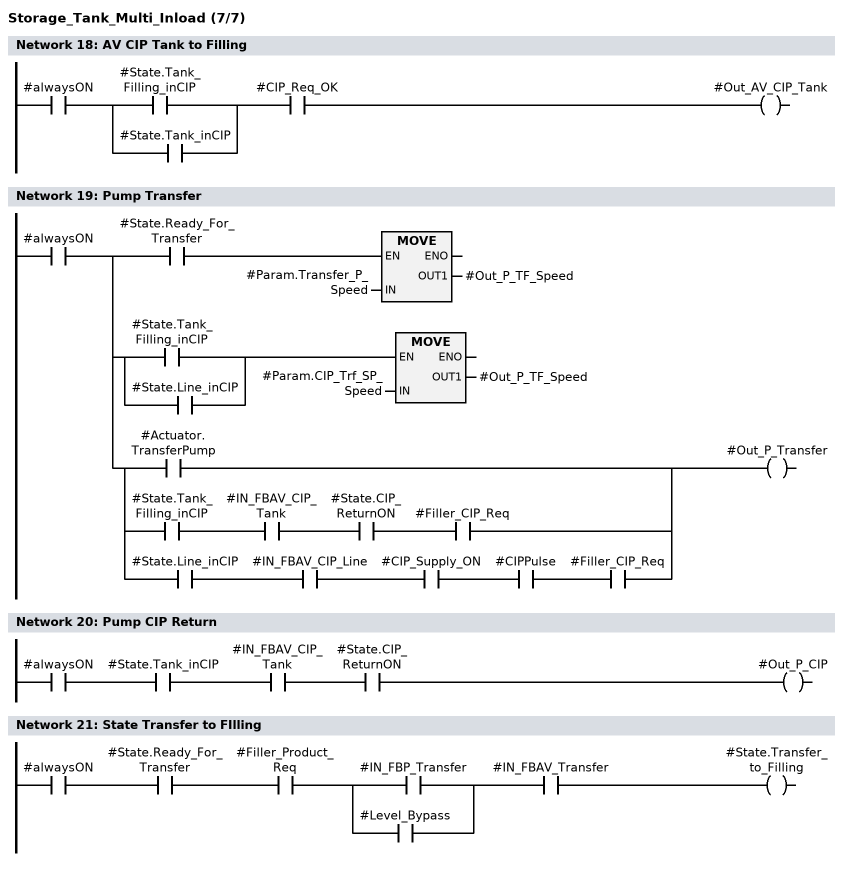
   RUNG wire#powerrail
      Contact( #alwaysON )
      wire#w1
      Contact( #State.Tank_Filling_inCIP )
      wire#w2
      Contact( #CIP_Req_OK )
      Coil( #Out_AV_CIP_Tank )
   END_RUNG
   RUNG wire#w1
      Contact( #State.Tank_inCIP )
   END_RUNG wire#w2
   // the same network as SCL:
   #Out_AV_CIP_Tank := #alwaysON AND (#State.Tank_Filling_inCIP OR #State.Tank_inCIP) AND #CIP_Req_OK;
END_REGION

REGION Network 19: Pump Transfer
   RUNG wire#powerrail
      Contact( #alwaysON )
      wire#w1
      Contact( #State.Ready_For_Transfer )
      Move(in := #Param.Transfer_P_Speed, out1 => #Out_P_TF_Speed)
   END_RUNG
   RUNG wire#w1
      Contact( #State.Tank_Filling_inCIP )
      wire#w2
      Move(in := #Param.CIP_Trf_SP_Speed, out1 => #Out_P_TF_Speed)
   END_RUNG
   RUNG wire#w1
      Contact( #State.Line_inCIP )
   END_RUNG wire#w2
   RUNG wire#w1
      Contact( #Actuator.TransferPump )
      wire#w3
      Coil( #Out_P_Transfer )
   END_RUNG
   RUNG wire#w1
      Contact( #State.Tank_Filling_inCIP )
      Contact( #IN_FBAV_CIP_Tank )
      Contact( #State.CIP_ReturnON )
      Contact( #Filler_CIP_Req )
   END_RUNG wire#w3
   RUNG wire#w1
      Contact( #State.Line_inCIP )
      Contact( #IN_FBAV_CIP_Line )
      Contact( #CIP_Supply_ON )
      Contact( #CIPPulse )
      Contact( #Filler_CIP_Req )
   END_RUNG wire#w3
   // the same network as SCL:
   IF #alwaysON AND #State.Ready_For_Transfer THEN #Out_P_TF_Speed := #Param.Transfer_P_Speed; END_IF;
   IF #alwaysON AND (#State.Tank_Filling_inCIP OR #State.Line_inCIP) THEN
       #Out_P_TF_Speed := #Param.CIP_Trf_SP_Speed;
   END_IF;
   #Out_P_Transfer := #alwaysON AND (#Actuator.TransferPump OR (#State.Tank_Filling_inCIP AND #IN_FBAV_CIP_Tank AND #State.CIP_ReturnON AND #Filler_CIP_Req) OR (#State.Line_inCIP AND #IN_FBAV_CIP_Line AND #CIP_Supply_ON AND #CIPPulse AND #Filler_CIP_Req));
END_REGION

REGION Network 20: Pump CIP Return
   RUNG wire#powerrail
      Contact( #alwaysON )
      Contact( #State.Tank_inCIP )
      Contact( #IN_FBAV_CIP_Tank )
      Contact( #State.CIP_ReturnON )
      Coil( #Out_P_CIP )
   END_RUNG
   // the same network as SCL:
   #Out_P_CIP := #alwaysON AND #State.Tank_inCIP AND #IN_FBAV_CIP_Tank AND #State.CIP_ReturnON;
END_REGION

REGION Network 21: State Transfer to FIlling
   RUNG wire#powerrail
      Contact( #alwaysON )
      Contact( #State.Ready_For_Transfer )
      Contact( #Filler_Product_Req )
      wire#w1
      Contact( #IN_FBP_Transfer )
      wire#w2
      Contact( #IN_FBAV_Transfer )
      Coil( #State.Transfer_to_Filling )
   END_RUNG
   RUNG wire#w1
      Contact( #Level_Bypass )
   END_RUNG wire#w2
   // the same network as SCL:
   #State.Transfer_to_Filling := #alwaysON AND #State.Ready_For_Transfer AND #Filler_Product_Req AND (#IN_FBP_Transfer OR #Level_Bypass) AND #IN_FBAV_Transfer;
END_REGION
END_FUNCTION_BLOCK

FUNCTION "Buffer" : Void   // FC11, LAD
{ S7_Optimized_Access := 'TRUE' }
VERSION : 0.1
// stored: AutoNumber true, IsIECCheckEnabled false, SetENOAutomatically false, UDAEnableTagReadback false
BEGIN

REGION Network 1: BFT 61 Rework 32
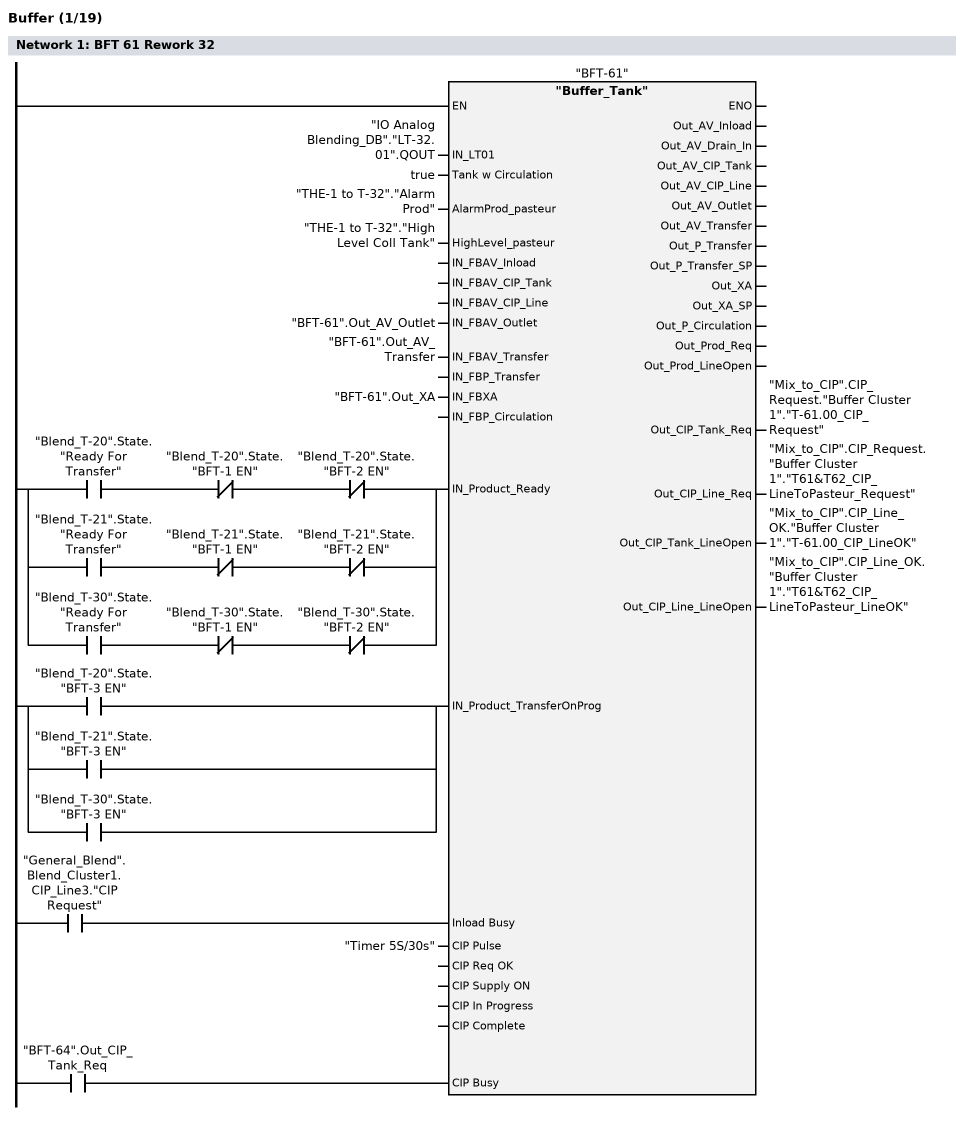
   RUNG wire#powerrail
      "BFT-61"(IN_Product_Ready := wire#w1, IN_Product_TransferOnProg := wire#w2, "Inload Busy" := wire#w3, "CIP Busy" := wire#w4, IN_LT01 := "IO Analog Blending_DB"."LT-32.01".QOUT, "Tank w Circulation" := true, AlarmProd_pasteur := "THE-1 to T-32"."Alarm Prod", HighLevel_pasteur := "THE-1 to T-32"."High Level Coll Tank", IN_FBAV_Inload :=, IN_FBAV_CIP_Tank :=, IN_FBAV_CIP_Line :=, IN_FBAV_Outlet := "BFT-61".Out_AV_Outlet, IN_FBAV_Transfer := "BFT-61".Out_AV_Transfer, IN_FBP_Transfer :=, IN_FBXA := "BFT-61".Out_XA, IN_FBP_Circulation :=, "CIP Pulse" := "Timer 5S/30s", "CIP Req OK" :=, "CIP Supply ON" :=, "CIP In Progress" :=, "CIP Complete" :=, Out_AV_Inload =>, Out_AV_Drain_In =>, Out_AV_CIP_Tank =>, Out_AV_CIP_Line =>, Out_AV_Outlet =>, Out_AV_Transfer =>, Out_P_Transfer =>, Out_P_Transfer_SP =>, Out_XA =>, Out_XA_SP =>, Out_P_Circulation =>, Out_Prod_Req =>, Out_Prod_LineOpen =>, Out_CIP_Tank_Req => "Mix_to_CIP".CIP_Request."Buffer Cluster 1"."T-61.00_CIP_Request", Out_CIP_Line_Req => "Mix_to_CIP".CIP_Request."Buffer Cluster 1"."T61&T62_CIP_LineToPasteur_Request", Out_CIP_Tank_LineOpen => "Mix_to_CIP".CIP_Line_OK."Buffer Cluster 1"."T-61.00_CIP_LineOK", Out_CIP_Line_LineOpen => "Mix_to_CIP".CIP_Line_OK."Buffer Cluster 1"."T61&T62_CIP_LineToPasteur_LineOK")
   END_RUNG
   RUNG wire#powerrail
      Contact( "Blend_T-20".State."Ready For Transfer" )
      I_Contact( "Blend_T-20".State."BFT-1 EN" )
      I_Contact( "Blend_T-20".State."BFT-2 EN" )
   END_RUNG wire#w1
   RUNG wire#powerrail
      Contact( "Blend_T-21".State."Ready For Transfer" )
      I_Contact( "Blend_T-21".State."BFT-1 EN" )
      I_Contact( "Blend_T-21".State."BFT-2 EN" )
   END_RUNG wire#w1
   RUNG wire#powerrail
      Contact( "Blend_T-30".State."Ready For Transfer" )
      I_Contact( "Blend_T-30".State."BFT-1 EN" )
      I_Contact( "Blend_T-30".State."BFT-2 EN" )
   END_RUNG wire#w1
   RUNG wire#powerrail
      Contact( "Blend_T-20".State."BFT-3 EN" )
   END_RUNG wire#w2
   RUNG wire#powerrail
      Contact( "Blend_T-21".State."BFT-3 EN" )
   END_RUNG wire#w2
   RUNG wire#powerrail
      Contact( "Blend_T-30".State."BFT-3 EN" )
   END_RUNG wire#w2
   RUNG wire#powerrail
      Contact( "General_Blend".Blend_Cluster1.CIP_Line3."CIP Request" )
   END_RUNG wire#w3
   RUNG wire#powerrail
      Contact( "BFT-64".Out_CIP_Tank_Req )
   END_RUNG wire#w4
   // the same network as SCL:
   "BFT-61"(IN_LT01 := "IO Analog Blending_DB"."LT-32.01".QOUT,   // "Buffer_Tank"
            "Tank w Circulation" := true,
            AlarmProd_pasteur := "THE-1 to T-32"."Alarm Prod",
            HighLevel_pasteur := "THE-1 to T-32"."High Level Coll Tank",
            IN_FBAV_Outlet := "BFT-61".Out_AV_Outlet,
            IN_FBAV_Transfer := "BFT-61".Out_AV_Transfer,
            IN_FBXA := "BFT-61".Out_XA,
            IN_Product_Ready := ("Blend_T-20".State."Ready For Transfer" AND NOT "Blend_T-20".State."BFT-1 EN" AND NOT "Blend_T-20".State."BFT-2 EN") OR ("Blend_T-21".State."Ready For Transfer" AND NOT "Blend_T-21".State."BFT-1 EN" AND NOT "Blend_T-21".State."BFT-2 EN") OR ("Blend_T-30".State."Ready For Transfer" AND NOT "Blend_T-30".State."BFT-1 EN" AND NOT "Blend_T-30".State."BFT-2 EN"),
            IN_Product_TransferOnProg := "Blend_T-20".State."BFT-3 EN" OR "Blend_T-21".State."BFT-3 EN" OR "Blend_T-30".State."BFT-3 EN",
            "Inload Busy" := "General_Blend".Blend_Cluster1.CIP_Line3."CIP Request",
            "CIP Pulse" := "Timer 5S/30s",
            "CIP Busy" := "BFT-64".Out_CIP_Tank_Req,
            Out_CIP_Tank_Req => "Mix_to_CIP".CIP_Request."Buffer Cluster 1"."T-61.00_CIP_Request",
            Out_CIP_Line_Req => "Mix_to_CIP".CIP_Request."Buffer Cluster 1"."T61&T62_CIP_LineToPasteur_Request",
            Out_CIP_Tank_LineOpen => "Mix_to_CIP".CIP_Line_OK."Buffer Cluster 1"."T-61.00_CIP_LineOK",
            Out_CIP_Line_LineOpen => "Mix_to_CIP".CIP_Line_OK."Buffer Cluster 1"."T61&T62_CIP_LineToPasteur_LineOK");
END_REGION

REGION Network 2: BFT 61 Feedback Instrument
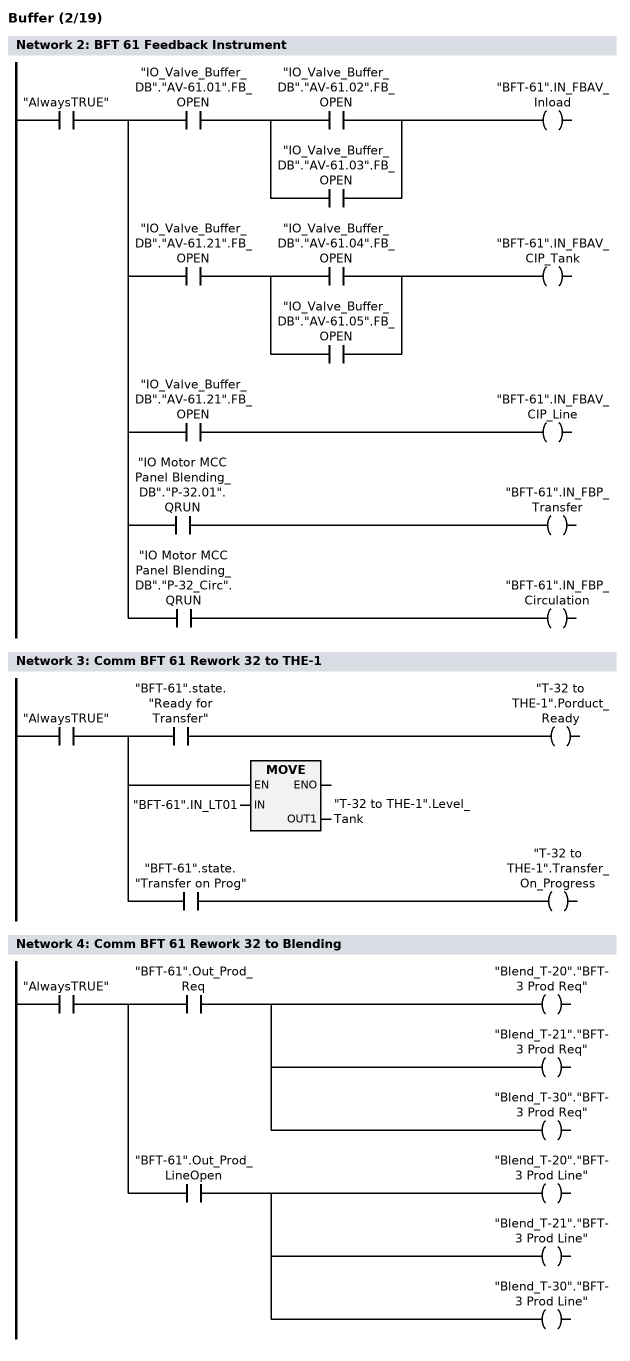
   RUNG wire#powerrail
      Contact( "AlwaysTRUE" )
      wire#w1
      Contact( "IO_Valve_Buffer_DB"."AV-61.01".FB_OPEN )
      wire#w2
      Contact( "IO_Valve_Buffer_DB"."AV-61.02".FB_OPEN )
      wire#w3
      Coil( "BFT-61".IN_FBAV_Inload )
   END_RUNG
   RUNG wire#w2
      Contact( "IO_Valve_Buffer_DB"."AV-61.03".FB_OPEN )
   END_RUNG wire#w3
   RUNG wire#w1
      Contact( "IO_Valve_Buffer_DB"."AV-61.21".FB_OPEN )
      wire#w4
      Contact( "IO_Valve_Buffer_DB"."AV-61.04".FB_OPEN )
      wire#w5
      Coil( "BFT-61".IN_FBAV_CIP_Tank )
   END_RUNG
   RUNG wire#w4
      Contact( "IO_Valve_Buffer_DB"."AV-61.05".FB_OPEN )
   END_RUNG wire#w5
   RUNG wire#w1
      Contact( "IO_Valve_Buffer_DB"."AV-61.21".FB_OPEN )
      Coil( "BFT-61".IN_FBAV_CIP_Line )
   END_RUNG
   RUNG wire#w1
      Contact( "IO Motor MCC Panel Blending_DB"."P-32.01".QRUN )
      Coil( "BFT-61".IN_FBP_Transfer )
   END_RUNG
   RUNG wire#w1
      Contact( "IO Motor MCC Panel Blending_DB"."P-32_Circ".QRUN )
      Coil( "BFT-61".IN_FBP_Circulation )
   END_RUNG
   // the same network as SCL:
   "BFT-61".IN_FBAV_Inload := "AlwaysTRUE" AND "IO_Valve_Buffer_DB"."AV-61.01".FB_OPEN AND ("IO_Valve_Buffer_DB"."AV-61.02".FB_OPEN OR "IO_Valve_Buffer_DB"."AV-61.03".FB_OPEN);
   "BFT-61".IN_FBAV_CIP_Tank := "AlwaysTRUE" AND "IO_Valve_Buffer_DB"."AV-61.21".FB_OPEN AND ("IO_Valve_Buffer_DB"."AV-61.04".FB_OPEN OR "IO_Valve_Buffer_DB"."AV-61.05".FB_OPEN);
   "BFT-61".IN_FBAV_CIP_Line := "AlwaysTRUE" AND "IO_Valve_Buffer_DB"."AV-61.21".FB_OPEN;
   "BFT-61".IN_FBP_Transfer := "AlwaysTRUE" AND "IO Motor MCC Panel Blending_DB"."P-32.01".QRUN;
   "BFT-61".IN_FBP_Circulation := "AlwaysTRUE" AND "IO Motor MCC Panel Blending_DB"."P-32_Circ".QRUN;
END_REGION

REGION Network 3: Comm BFT 61 Rework 32 to THE-1
   RUNG wire#powerrail
      Contact( "AlwaysTRUE" )
      wire#w1
      Contact( "BFT-61".state."Ready for Transfer" )
      Coil( "T-32 to THE-1".Porduct_Ready )
   END_RUNG
   RUNG wire#w1
      Move(in := "BFT-61".IN_LT01, out1 => "T-32 to THE-1".Level_Tank)
   END_RUNG
   RUNG wire#w1
      Contact( "BFT-61".state."Transfer on Prog" )
      Coil( "T-32 to THE-1".Transfer_On_Progress )
   END_RUNG
   // the same network as SCL:
   "T-32 to THE-1".Porduct_Ready := "AlwaysTRUE" AND "BFT-61".state."Ready for Transfer";
   IF "AlwaysTRUE" THEN "T-32 to THE-1".Level_Tank := "BFT-61".IN_LT01; END_IF;
   "T-32 to THE-1".Transfer_On_Progress := "AlwaysTRUE" AND "BFT-61".state."Transfer on Prog";
END_REGION

REGION Network 4: Comm BFT 61 Rework 32 to Blending
   RUNG wire#powerrail
      Contact( "AlwaysTRUE" )
      wire#w1
      Contact( "BFT-61".Out_Prod_Req )
      wire#w2
      Coil( "Blend_T-20"."BFT-3 Prod Req" )
   END_RUNG
   RUNG wire#w2
      Coil( "Blend_T-21"."BFT-3 Prod Req" )
   END_RUNG
   RUNG wire#w2
      Coil( "Blend_T-30"."BFT-3 Prod Req" )
   END_RUNG
   RUNG wire#w1
      Contact( "BFT-61".Out_Prod_LineOpen )
      wire#w3
      Coil( "Blend_T-20"."BFT-3 Prod Line" )
   END_RUNG
   RUNG wire#w3
      Coil( "Blend_T-21"."BFT-3 Prod Line" )
   END_RUNG
   RUNG wire#w3
      Coil( "Blend_T-30"."BFT-3 Prod Line" )
   END_RUNG
   // the same network as SCL:
   "Blend_T-20"."BFT-3 Prod Req" := "AlwaysTRUE" AND "BFT-61".Out_Prod_Req;
   "Blend_T-21"."BFT-3 Prod Req" := "Blend_T-20"."BFT-3 Prod Req";
   "Blend_T-30"."BFT-3 Prod Req" := "Blend_T-20"."BFT-3 Prod Req";
   "Blend_T-20"."BFT-3 Prod Line" := "AlwaysTRUE" AND "BFT-61".Out_Prod_LineOpen;
   "Blend_T-21"."BFT-3 Prod Line" := "Blend_T-20"."BFT-3 Prod Line";
   "Blend_T-30"."BFT-3 Prod Line" := "Blend_T-20"."BFT-3 Prod Line";
END_REGION

REGION Network 6: BFT 64 Rework 22
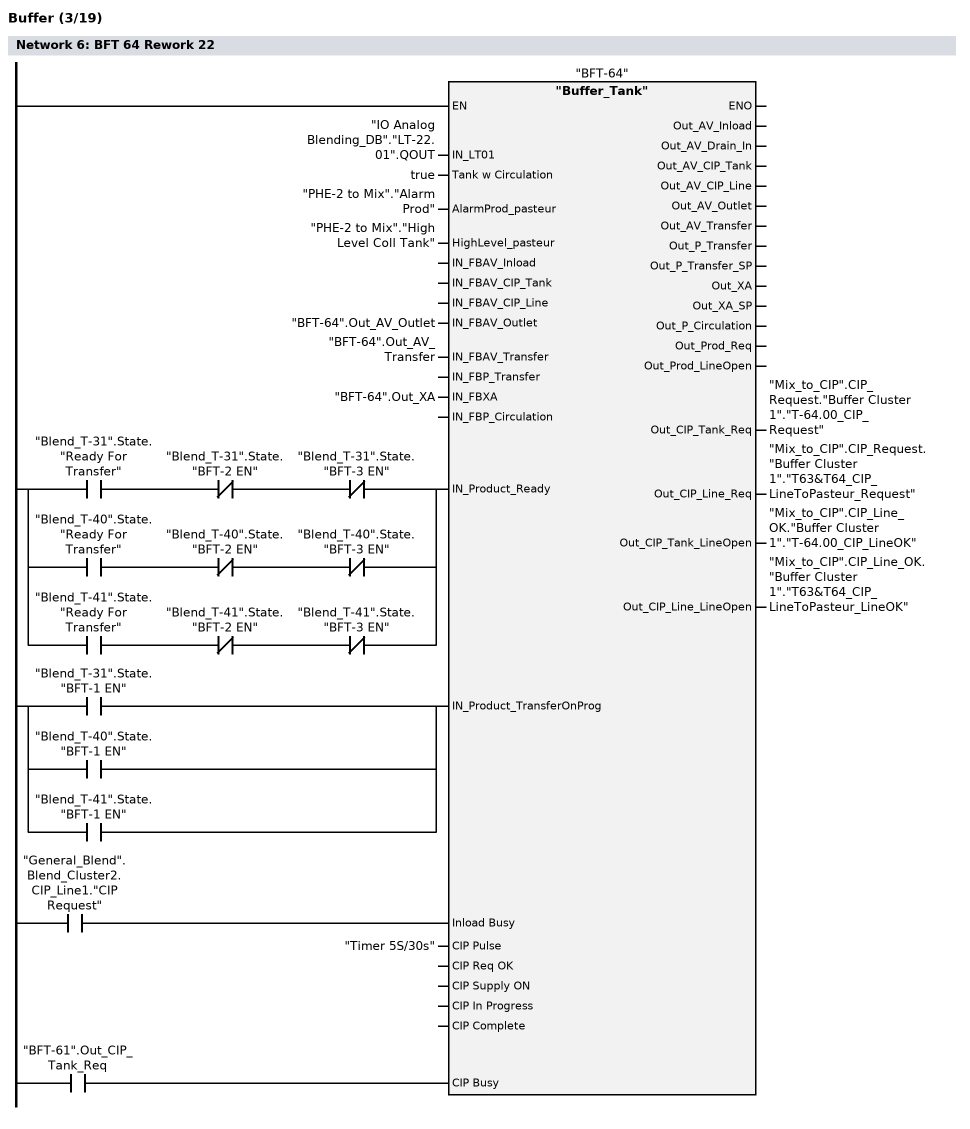
   RUNG wire#powerrail
      "BFT-64"(IN_Product_Ready := wire#w1, IN_Product_TransferOnProg := wire#w2, "Inload Busy" := wire#w3, "CIP Busy" := wire#w4, IN_LT01 := "IO Analog Blending_DB"."LT-22.01".QOUT, "Tank w Circulation" := true, AlarmProd_pasteur := "PHE-2 to Mix"."Alarm Prod", HighLevel_pasteur := "PHE-2 to Mix"."High Level Coll Tank", IN_FBAV_Inload :=, IN_FBAV_CIP_Tank :=, IN_FBAV_CIP_Line :=, IN_FBAV_Outlet := "BFT-64".Out_AV_Outlet, IN_FBAV_Transfer := "BFT-64".Out_AV_Transfer, IN_FBP_Transfer :=, IN_FBXA := "BFT-64".Out_XA, IN_FBP_Circulation :=, "CIP Pulse" := "Timer 5S/30s", "CIP Req OK" :=, "CIP Supply ON" :=, "CIP In Progress" :=, "CIP Complete" :=, Out_AV_Inload =>, Out_AV_Drain_In =>, Out_AV_CIP_Tank =>, Out_AV_CIP_Line =>, Out_AV_Outlet =>, Out_AV_Transfer =>, Out_P_Transfer =>, Out_P_Transfer_SP =>, Out_XA =>, Out_XA_SP =>, Out_P_Circulation =>, Out_Prod_Req =>, Out_Prod_LineOpen =>, Out_CIP_Tank_Req => "Mix_to_CIP".CIP_Request."Buffer Cluster 1"."T-64.00_CIP_Request", Out_CIP_Line_Req => "Mix_to_CIP".CIP_Request."Buffer Cluster 1"."T63&T64_CIP_LineToPasteur_Request", Out_CIP_Tank_LineOpen => "Mix_to_CIP".CIP_Line_OK."Buffer Cluster 1"."T-64.00_CIP_LineOK", Out_CIP_Line_LineOpen => "Mix_to_CIP".CIP_Line_OK."Buffer Cluster 1"."T63&T64_CIP_LineToPasteur_LineOK")
   END_RUNG
   RUNG wire#powerrail
      Contact( "Blend_T-31".State."Ready For Transfer" )
      I_Contact( "Blend_T-31".State."BFT-2 EN" )
      I_Contact( "Blend_T-31".State."BFT-3 EN" )
   END_RUNG wire#w1
   RUNG wire#powerrail
      Contact( "Blend_T-40".State."Ready For Transfer" )
      I_Contact( "Blend_T-40".State."BFT-2 EN" )
      I_Contact( "Blend_T-40".State."BFT-3 EN" )
   END_RUNG wire#w1
   RUNG wire#powerrail
      Contact( "Blend_T-41".State."Ready For Transfer" )
      I_Contact( "Blend_T-41".State."BFT-2 EN" )
      I_Contact( "Blend_T-41".State."BFT-3 EN" )
   END_RUNG wire#w1
   RUNG wire#powerrail
      Contact( "Blend_T-31".State."BFT-1 EN" )
   END_RUNG wire#w2
   RUNG wire#powerrail
      Contact( "Blend_T-40".State."BFT-1 EN" )
   END_RUNG wire#w2
   RUNG wire#powerrail
      Contact( "Blend_T-41".State."BFT-1 EN" )
   END_RUNG wire#w2
   RUNG wire#powerrail
      Contact( "General_Blend".Blend_Cluster2.CIP_Line1."CIP Request" )
   END_RUNG wire#w3
   RUNG wire#powerrail
      Contact( "BFT-61".Out_CIP_Tank_Req )
   END_RUNG wire#w4
   // the same network as SCL:
   "BFT-64"(IN_LT01 := "IO Analog Blending_DB"."LT-22.01".QOUT,   // "Buffer_Tank"
            "Tank w Circulation" := true,
            AlarmProd_pasteur := "PHE-2 to Mix"."Alarm Prod",
            HighLevel_pasteur := "PHE-2 to Mix"."High Level Coll Tank",
            IN_FBAV_Outlet := "BFT-64".Out_AV_Outlet,
            IN_FBAV_Transfer := "BFT-64".Out_AV_Transfer,
            IN_FBXA := "BFT-64".Out_XA,
            IN_Product_Ready := ("Blend_T-31".State."Ready For Transfer" AND NOT "Blend_T-31".State."BFT-2 EN" AND NOT "Blend_T-31".State."BFT-3 EN") OR ("Blend_T-40".State."Ready For Transfer" AND NOT "Blend_T-40".State."BFT-2 EN" AND NOT "Blend_T-40".State."BFT-3 EN") OR ("Blend_T-41".State."Ready For Transfer" AND NOT "Blend_T-41".State."BFT-2 EN" AND NOT "Blend_T-41".State."BFT-3 EN"),
            IN_Product_TransferOnProg := "Blend_T-31".State."BFT-1 EN" OR "Blend_T-40".State."BFT-1 EN" OR "Blend_T-41".State."BFT-1 EN",
            "Inload Busy" := "General_Blend".Blend_Cluster2.CIP_Line1."CIP Request",
            "CIP Pulse" := "Timer 5S/30s",
            "CIP Busy" := "BFT-61".Out_CIP_Tank_Req,
            Out_CIP_Tank_Req => "Mix_to_CIP".CIP_Request."Buffer Cluster 1"."T-64.00_CIP_Request",
            Out_CIP_Line_Req => "Mix_to_CIP".CIP_Request."Buffer Cluster 1"."T63&T64_CIP_LineToPasteur_Request",
            Out_CIP_Tank_LineOpen => "Mix_to_CIP".CIP_Line_OK."Buffer Cluster 1"."T-64.00_CIP_LineOK",
            Out_CIP_Line_LineOpen => "Mix_to_CIP".CIP_Line_OK."Buffer Cluster 1"."T63&T64_CIP_LineToPasteur_LineOK");
END_REGION

REGION Network 7: BFT 64 Feedback Instrument
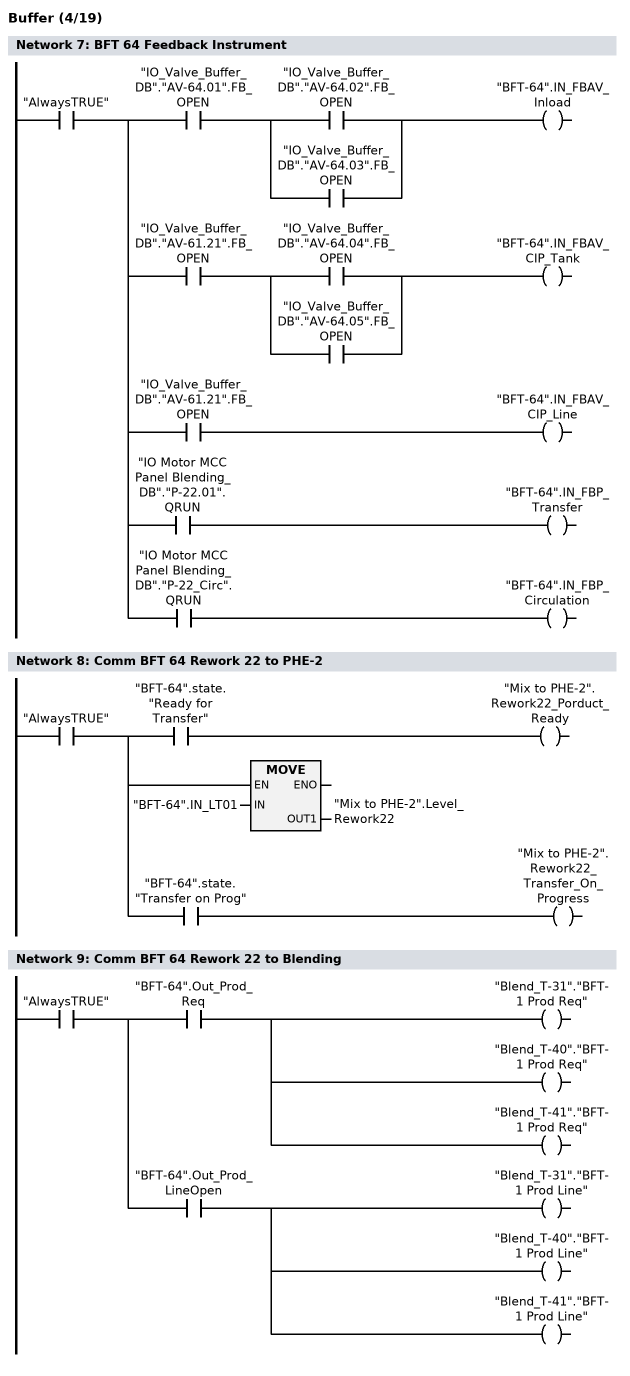
   RUNG wire#powerrail
      Contact( "AlwaysTRUE" )
      wire#w1
      Contact( "IO_Valve_Buffer_DB"."AV-64.01".FB_OPEN )
      wire#w2
      Contact( "IO_Valve_Buffer_DB"."AV-64.02".FB_OPEN )
      wire#w3
      Coil( "BFT-64".IN_FBAV_Inload )
   END_RUNG
   RUNG wire#w2
      Contact( "IO_Valve_Buffer_DB"."AV-64.03".FB_OPEN )
   END_RUNG wire#w3
   RUNG wire#w1
      Contact( "IO_Valve_Buffer_DB"."AV-61.21".FB_OPEN )
      wire#w4
      Contact( "IO_Valve_Buffer_DB"."AV-64.04".FB_OPEN )
      wire#w5
      Coil( "BFT-64".IN_FBAV_CIP_Tank )
   END_RUNG
   RUNG wire#w4
      Contact( "IO_Valve_Buffer_DB"."AV-64.05".FB_OPEN )
   END_RUNG wire#w5
   RUNG wire#w1
      Contact( "IO_Valve_Buffer_DB"."AV-61.21".FB_OPEN )
      Coil( "BFT-64".IN_FBAV_CIP_Line )
   END_RUNG
   RUNG wire#w1
      Contact( "IO Motor MCC Panel Blending_DB"."P-22.01".QRUN )
      Coil( "BFT-64".IN_FBP_Transfer )
   END_RUNG
   RUNG wire#w1
      Contact( "IO Motor MCC Panel Blending_DB"."P-22_Circ".QRUN )
      Coil( "BFT-64".IN_FBP_Circulation )
   END_RUNG
   // the same network as SCL:
   "BFT-64".IN_FBAV_Inload := "AlwaysTRUE" AND "IO_Valve_Buffer_DB"."AV-64.01".FB_OPEN AND ("IO_Valve_Buffer_DB"."AV-64.02".FB_OPEN OR "IO_Valve_Buffer_DB"."AV-64.03".FB_OPEN);
   "BFT-64".IN_FBAV_CIP_Tank := "AlwaysTRUE" AND "IO_Valve_Buffer_DB"."AV-61.21".FB_OPEN AND ("IO_Valve_Buffer_DB"."AV-64.04".FB_OPEN OR "IO_Valve_Buffer_DB"."AV-64.05".FB_OPEN);
   "BFT-64".IN_FBAV_CIP_Line := "AlwaysTRUE" AND "IO_Valve_Buffer_DB"."AV-61.21".FB_OPEN;
   "BFT-64".IN_FBP_Transfer := "AlwaysTRUE" AND "IO Motor MCC Panel Blending_DB"."P-22.01".QRUN;
   "BFT-64".IN_FBP_Circulation := "AlwaysTRUE" AND "IO Motor MCC Panel Blending_DB"."P-22_Circ".QRUN;
END_REGION

REGION Network 8: Comm BFT 64 Rework 22 to PHE-2
   RUNG wire#powerrail
      Contact( "AlwaysTRUE" )
      wire#w1
      Contact( "BFT-64".state."Ready for Transfer" )
      Coil( "Mix to PHE-2".Rework22_Porduct_Ready )
   END_RUNG
   RUNG wire#w1
      Move(in := "BFT-64".IN_LT01, out1 => "Mix to PHE-2".Level_Rework22)
   END_RUNG
   RUNG wire#w1
      Contact( "BFT-64".state."Transfer on Prog" )
      Coil( "Mix to PHE-2".Rework22_Transfer_On_Progress )
   END_RUNG
   // the same network as SCL:
   "Mix to PHE-2".Rework22_Porduct_Ready := "AlwaysTRUE" AND "BFT-64".state."Ready for Transfer";
   IF "AlwaysTRUE" THEN "Mix to PHE-2".Level_Rework22 := "BFT-64".IN_LT01; END_IF;
   "Mix to PHE-2".Rework22_Transfer_On_Progress := "AlwaysTRUE" AND "BFT-64".state."Transfer on Prog";
END_REGION

REGION Network 9: Comm BFT 64 Rework 22 to Blending
   RUNG wire#powerrail
      Contact( "AlwaysTRUE" )
      wire#w1
      Contact( "BFT-64".Out_Prod_Req )
      wire#w2
      Coil( "Blend_T-31"."BFT-1 Prod Req" )
   END_RUNG
   RUNG wire#w2
      Coil( "Blend_T-40"."BFT-1 Prod Req" )
   END_RUNG
   RUNG wire#w2
      Coil( "Blend_T-41"."BFT-1 Prod Req" )
   END_RUNG
   RUNG wire#w1
      Contact( "BFT-64".Out_Prod_LineOpen )
      wire#w3
      Coil( "Blend_T-31"."BFT-1 Prod Line" )
   END_RUNG
   RUNG wire#w3
      Coil( "Blend_T-40"."BFT-1 Prod Line" )
   END_RUNG
   RUNG wire#w3
      Coil( "Blend_T-41"."BFT-1 Prod Line" )
   END_RUNG
   // the same network as SCL:
   "Blend_T-31"."BFT-1 Prod Req" := "AlwaysTRUE" AND "BFT-64".Out_Prod_Req;
   "Blend_T-40"."BFT-1 Prod Req" := "Blend_T-31"."BFT-1 Prod Req";
   "Blend_T-41"."BFT-1 Prod Req" := "Blend_T-31"."BFT-1 Prod Req";
   "Blend_T-31"."BFT-1 Prod Line" := "AlwaysTRUE" AND "BFT-64".Out_Prod_LineOpen;
   "Blend_T-40"."BFT-1 Prod Line" := "Blend_T-31"."BFT-1 Prod Line";
   "Blend_T-41"."BFT-1 Prod Line" := "Blend_T-31"."BFT-1 Prod Line";
END_REGION

REGION Network 11: BFT 65
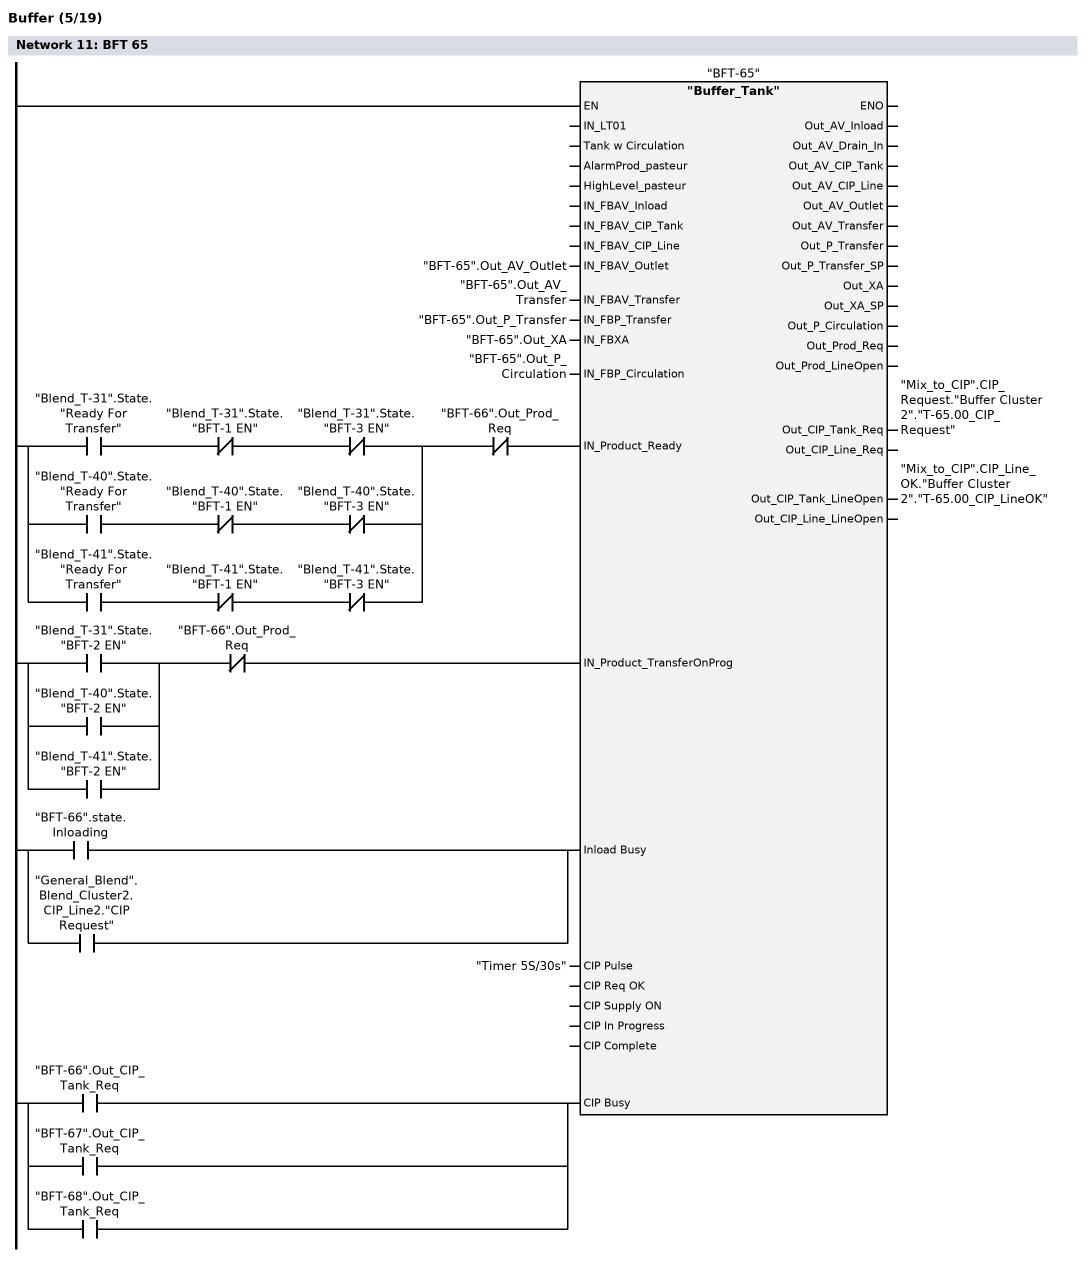
   RUNG wire#powerrail
      "BFT-65"(IN_Product_Ready := wire#w2, IN_Product_TransferOnProg := wire#w4, "Inload Busy" := wire#w5, "CIP Busy" := wire#w6, IN_LT01 :=, "Tank w Circulation" :=, AlarmProd_pasteur :=, HighLevel_pasteur :=, IN_FBAV_Inload :=, IN_FBAV_CIP_Tank :=, IN_FBAV_CIP_Line :=, IN_FBAV_Outlet := "BFT-65".Out_AV_Outlet, IN_FBAV_Transfer := "BFT-65".Out_AV_Transfer, IN_FBP_Transfer := "BFT-65".Out_P_Transfer, IN_FBXA := "BFT-65".Out_XA, IN_FBP_Circulation := "BFT-65".Out_P_Circulation, "CIP Pulse" := "Timer 5S/30s", "CIP Req OK" :=, "CIP Supply ON" :=, "CIP In Progress" :=, "CIP Complete" :=, Out_AV_Inload =>, Out_AV_Drain_In =>, Out_AV_CIP_Tank =>, Out_AV_CIP_Line =>, Out_AV_Outlet =>, Out_AV_Transfer =>, Out_P_Transfer =>, Out_P_Transfer_SP =>, Out_XA =>, Out_XA_SP =>, Out_P_Circulation =>, Out_Prod_Req =>, Out_Prod_LineOpen =>, Out_CIP_Tank_Req => "Mix_to_CIP".CIP_Request."Buffer Cluster 2"."T-65.00_CIP_Request", Out_CIP_Line_Req =>, Out_CIP_Tank_LineOpen => "Mix_to_CIP".CIP_Line_OK."Buffer Cluster 2"."T-65.00_CIP_LineOK", Out_CIP_Line_LineOpen =>)
   END_RUNG
   RUNG wire#powerrail
      Contact( "Blend_T-31".State."Ready For Transfer" )
      I_Contact( "Blend_T-31".State."BFT-1 EN" )
      I_Contact( "Blend_T-31".State."BFT-3 EN" )
      wire#w1
      I_Contact( "BFT-66".Out_Prod_Req )
   END_RUNG wire#w2
   RUNG wire#powerrail
      Contact( "Blend_T-40".State."Ready For Transfer" )
      I_Contact( "Blend_T-40".State."BFT-1 EN" )
      I_Contact( "Blend_T-40".State."BFT-3 EN" )
   END_RUNG wire#w1
   RUNG wire#powerrail
      Contact( "Blend_T-41".State."Ready For Transfer" )
      I_Contact( "Blend_T-41".State."BFT-1 EN" )
      I_Contact( "Blend_T-41".State."BFT-3 EN" )
   END_RUNG wire#w1
   RUNG wire#powerrail
      Contact( "Blend_T-31".State."BFT-2 EN" )
      wire#w3
      I_Contact( "BFT-66".Out_Prod_Req )
   END_RUNG wire#w4
   RUNG wire#powerrail
      Contact( "Blend_T-40".State."BFT-2 EN" )
   END_RUNG wire#w3
   RUNG wire#powerrail
      Contact( "Blend_T-41".State."BFT-2 EN" )
   END_RUNG wire#w3
   RUNG wire#powerrail
      Contact( "BFT-66".state.Inloading )
   END_RUNG wire#w5
   RUNG wire#powerrail
      Contact( "General_Blend".Blend_Cluster2.CIP_Line2."CIP Request" )
   END_RUNG wire#w5
   RUNG wire#powerrail
      Contact( "BFT-66".Out_CIP_Tank_Req )
   END_RUNG wire#w6
   RUNG wire#powerrail
      Contact( "BFT-67".Out_CIP_Tank_Req )
   END_RUNG wire#w6
   RUNG wire#powerrail
      Contact( "BFT-68".Out_CIP_Tank_Req )
   END_RUNG wire#w6
   // the same network as SCL:
   "BFT-65"(IN_FBAV_Outlet := "BFT-65".Out_AV_Outlet,   // "Buffer_Tank"
            IN_FBAV_Transfer := "BFT-65".Out_AV_Transfer,
            IN_FBP_Transfer := "BFT-65".Out_P_Transfer,
            IN_FBXA := "BFT-65".Out_XA,
            IN_FBP_Circulation := "BFT-65".Out_P_Circulation,
            IN_Product_Ready := (("Blend_T-31".State."Ready For Transfer" AND NOT "Blend_T-31".State."BFT-1 EN" AND NOT "Blend_T-31".State."BFT-3 EN") OR ("Blend_T-40".State."Ready For Transfer" AND NOT "Blend_T-40".State."BFT-1 EN" AND NOT "Blend_T-40".State."BFT-3 EN") OR ("Blend_T-41".State."Ready For Transfer" AND NOT "Blend_T-41".State."BFT-1 EN" AND NOT "Blend_T-41".State."BFT-3 EN")) AND NOT "BFT-66".Out_Prod_Req,
            IN_Product_TransferOnProg := ("Blend_T-31".State."BFT-2 EN" OR "Blend_T-40".State."BFT-2 EN" OR "Blend_T-41".State."BFT-2 EN") AND NOT "BFT-66".Out_Prod_Req,
            "Inload Busy" := "BFT-66".state.Inloading OR "General_Blend".Blend_Cluster2.CIP_Line2."CIP Request",
            "CIP Pulse" := "Timer 5S/30s",
            "CIP Busy" := "BFT-66".Out_CIP_Tank_Req OR "BFT-67".Out_CIP_Tank_Req OR "BFT-68".Out_CIP_Tank_Req,
            Out_CIP_Tank_Req => "Mix_to_CIP".CIP_Request."Buffer Cluster 2"."T-65.00_CIP_Request",
            Out_CIP_Tank_LineOpen => "Mix_to_CIP".CIP_Line_OK."Buffer Cluster 2"."T-65.00_CIP_LineOK");
END_REGION

REGION Network 12: BFT 65 Feedback Instrument
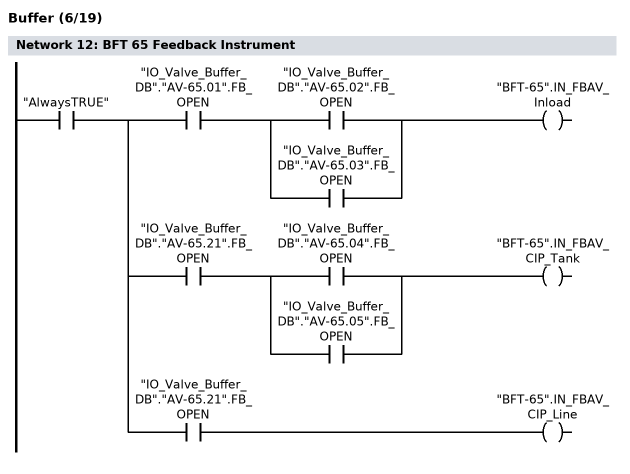
   RUNG wire#powerrail
      Contact( "AlwaysTRUE" )
      wire#w1
      Contact( "IO_Valve_Buffer_DB"."AV-65.01".FB_OPEN )
      wire#w2
      Contact( "IO_Valve_Buffer_DB"."AV-65.02".FB_OPEN )
      wire#w3
      Coil( "BFT-65".IN_FBAV_Inload )
   END_RUNG
   RUNG wire#w2
      Contact( "IO_Valve_Buffer_DB"."AV-65.03".FB_OPEN )
   END_RUNG wire#w3
   RUNG wire#w1
      Contact( "IO_Valve_Buffer_DB"."AV-65.21".FB_OPEN )
      wire#w4
      Contact( "IO_Valve_Buffer_DB"."AV-65.04".FB_OPEN )
      wire#w5
      Coil( "BFT-65".IN_FBAV_CIP_Tank )
   END_RUNG
   RUNG wire#w4
      Contact( "IO_Valve_Buffer_DB"."AV-65.05".FB_OPEN )
   END_RUNG wire#w5
   RUNG wire#w1
      Contact( "IO_Valve_Buffer_DB"."AV-65.21".FB_OPEN )
      Coil( "BFT-65".IN_FBAV_CIP_Line )
   END_RUNG
   // the same network as SCL:
   "BFT-65".IN_FBAV_Inload := "AlwaysTRUE" AND "IO_Valve_Buffer_DB"."AV-65.01".FB_OPEN AND ("IO_Valve_Buffer_DB"."AV-65.02".FB_OPEN OR "IO_Valve_Buffer_DB"."AV-65.03".FB_OPEN);
   "BFT-65".IN_FBAV_CIP_Tank := "AlwaysTRUE" AND "IO_Valve_Buffer_DB"."AV-65.21".FB_OPEN AND ("IO_Valve_Buffer_DB"."AV-65.04".FB_OPEN OR "IO_Valve_Buffer_DB"."AV-65.05".FB_OPEN);
   "BFT-65".IN_FBAV_CIP_Line := "AlwaysTRUE" AND "IO_Valve_Buffer_DB"."AV-65.21".FB_OPEN;
END_REGION

REGION Network 13: BFT 66
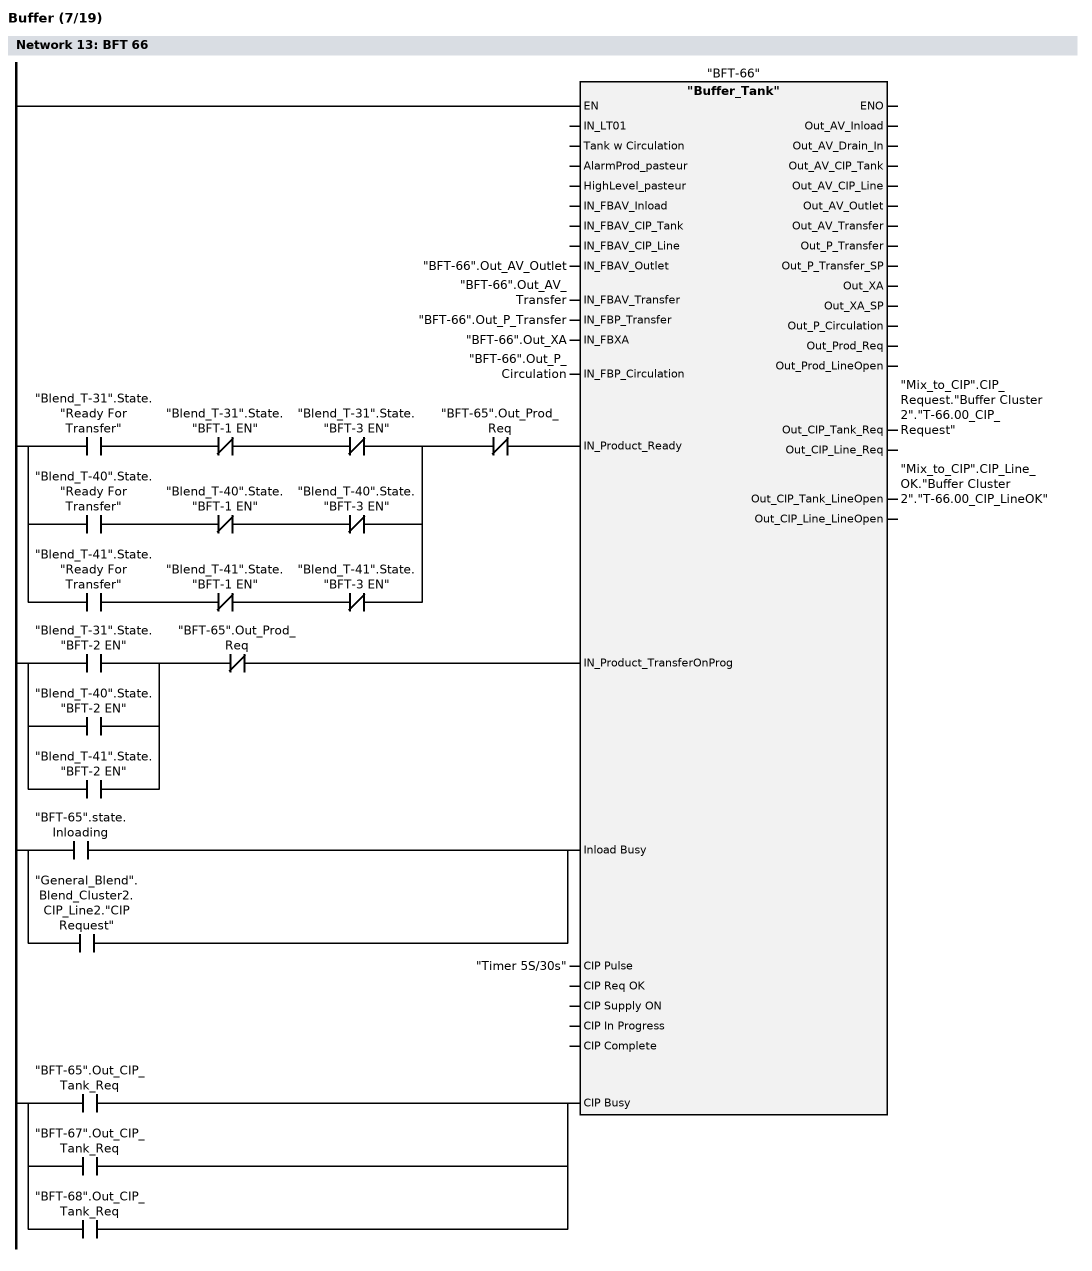
   RUNG wire#powerrail
      "BFT-66"(IN_Product_Ready := wire#w2, IN_Product_TransferOnProg := wire#w4, "Inload Busy" := wire#w5, "CIP Busy" := wire#w6, IN_LT01 :=, "Tank w Circulation" :=, AlarmProd_pasteur :=, HighLevel_pasteur :=, IN_FBAV_Inload :=, IN_FBAV_CIP_Tank :=, IN_FBAV_CIP_Line :=, IN_FBAV_Outlet := "BFT-66".Out_AV_Outlet, IN_FBAV_Transfer := "BFT-66".Out_AV_Transfer, IN_FBP_Transfer := "BFT-66".Out_P_Transfer, IN_FBXA := "BFT-66".Out_XA, IN_FBP_Circulation := "BFT-66".Out_P_Circulation, "CIP Pulse" := "Timer 5S/30s", "CIP Req OK" :=, "CIP Supply ON" :=, "CIP In Progress" :=, "CIP Complete" :=, Out_AV_Inload =>, Out_AV_Drain_In =>, Out_AV_CIP_Tank =>, Out_AV_CIP_Line =>, Out_AV_Outlet =>, Out_AV_Transfer =>, Out_P_Transfer =>, Out_P_Transfer_SP =>, Out_XA =>, Out_XA_SP =>, Out_P_Circulation =>, Out_Prod_Req =>, Out_Prod_LineOpen =>, Out_CIP_Tank_Req => "Mix_to_CIP".CIP_Request."Buffer Cluster 2"."T-66.00_CIP_Request", Out_CIP_Line_Req =>, Out_CIP_Tank_LineOpen => "Mix_to_CIP".CIP_Line_OK."Buffer Cluster 2"."T-66.00_CIP_LineOK", Out_CIP_Line_LineOpen =>)
   END_RUNG
   RUNG wire#powerrail
      Contact( "Blend_T-31".State."Ready For Transfer" )
      I_Contact( "Blend_T-31".State."BFT-1 EN" )
      I_Contact( "Blend_T-31".State."BFT-3 EN" )
      wire#w1
      I_Contact( "BFT-65".Out_Prod_Req )
   END_RUNG wire#w2
   RUNG wire#powerrail
      Contact( "Blend_T-40".State."Ready For Transfer" )
      I_Contact( "Blend_T-40".State."BFT-1 EN" )
      I_Contact( "Blend_T-40".State."BFT-3 EN" )
   END_RUNG wire#w1
   RUNG wire#powerrail
      Contact( "Blend_T-41".State."Ready For Transfer" )
      I_Contact( "Blend_T-41".State."BFT-1 EN" )
      I_Contact( "Blend_T-41".State."BFT-3 EN" )
   END_RUNG wire#w1
   RUNG wire#powerrail
      Contact( "Blend_T-31".State."BFT-2 EN" )
      wire#w3
      I_Contact( "BFT-65".Out_Prod_Req )
   END_RUNG wire#w4
   RUNG wire#powerrail
      Contact( "Blend_T-40".State."BFT-2 EN" )
   END_RUNG wire#w3
   RUNG wire#powerrail
      Contact( "Blend_T-41".State."BFT-2 EN" )
   END_RUNG wire#w3
   RUNG wire#powerrail
      Contact( "BFT-65".state.Inloading )
   END_RUNG wire#w5
   RUNG wire#powerrail
      Contact( "General_Blend".Blend_Cluster2.CIP_Line2."CIP Request" )
   END_RUNG wire#w5
   RUNG wire#powerrail
      Contact( "BFT-65".Out_CIP_Tank_Req )
   END_RUNG wire#w6
   RUNG wire#powerrail
      Contact( "BFT-67".Out_CIP_Tank_Req )
   END_RUNG wire#w6
   RUNG wire#powerrail
      Contact( "BFT-68".Out_CIP_Tank_Req )
   END_RUNG wire#w6
   // the same network as SCL:
   "BFT-66"(IN_FBAV_Outlet := "BFT-66".Out_AV_Outlet,   // "Buffer_Tank"
            IN_FBAV_Transfer := "BFT-66".Out_AV_Transfer,
            IN_FBP_Transfer := "BFT-66".Out_P_Transfer,
            IN_FBXA := "BFT-66".Out_XA,
            IN_FBP_Circulation := "BFT-66".Out_P_Circulation,
            IN_Product_Ready := (("Blend_T-31".State."Ready For Transfer" AND NOT "Blend_T-31".State."BFT-1 EN" AND NOT "Blend_T-31".State."BFT-3 EN") OR ("Blend_T-40".State."Ready For Transfer" AND NOT "Blend_T-40".State."BFT-1 EN" AND NOT "Blend_T-40".State."BFT-3 EN") OR ("Blend_T-41".State."Ready For Transfer" AND NOT "Blend_T-41".State."BFT-1 EN" AND NOT "Blend_T-41".State."BFT-3 EN")) AND NOT "BFT-65".Out_Prod_Req,
            IN_Product_TransferOnProg := ("Blend_T-31".State."BFT-2 EN" OR "Blend_T-40".State."BFT-2 EN" OR "Blend_T-41".State."BFT-2 EN") AND NOT "BFT-65".Out_Prod_Req,
            "Inload Busy" := "BFT-65".state.Inloading OR "General_Blend".Blend_Cluster2.CIP_Line2."CIP Request",
            "CIP Pulse" := "Timer 5S/30s",
            "CIP Busy" := "BFT-65".Out_CIP_Tank_Req OR "BFT-67".Out_CIP_Tank_Req OR "BFT-68".Out_CIP_Tank_Req,
            Out_CIP_Tank_Req => "Mix_to_CIP".CIP_Request."Buffer Cluster 2"."T-66.00_CIP_Request",
            Out_CIP_Tank_LineOpen => "Mix_to_CIP".CIP_Line_OK."Buffer Cluster 2"."T-66.00_CIP_LineOK");
END_REGION

REGION Network 14: BFT 66 Feedback Instrument
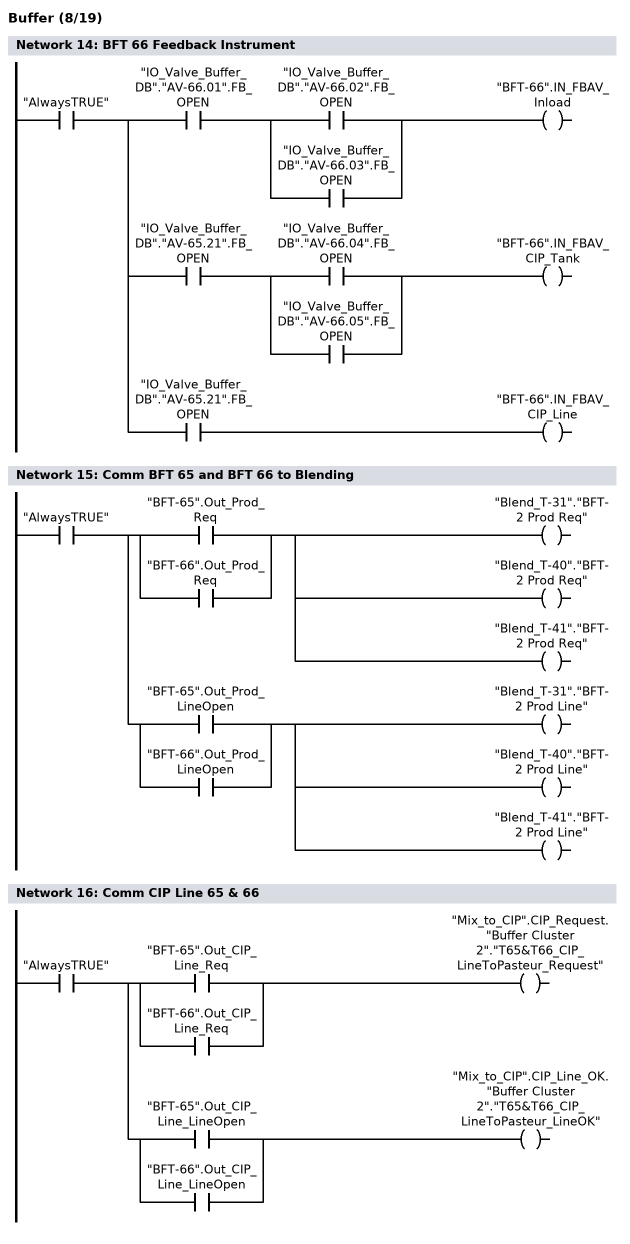
   RUNG wire#powerrail
      Contact( "AlwaysTRUE" )
      wire#w1
      Contact( "IO_Valve_Buffer_DB"."AV-66.01".FB_OPEN )
      wire#w2
      Contact( "IO_Valve_Buffer_DB"."AV-66.02".FB_OPEN )
      wire#w3
      Coil( "BFT-66".IN_FBAV_Inload )
   END_RUNG
   RUNG wire#w2
      Contact( "IO_Valve_Buffer_DB"."AV-66.03".FB_OPEN )
   END_RUNG wire#w3
   RUNG wire#w1
      Contact( "IO_Valve_Buffer_DB"."AV-65.21".FB_OPEN )
      wire#w4
      Contact( "IO_Valve_Buffer_DB"."AV-66.04".FB_OPEN )
      wire#w5
      Coil( "BFT-66".IN_FBAV_CIP_Tank )
   END_RUNG
   RUNG wire#w4
      Contact( "IO_Valve_Buffer_DB"."AV-66.05".FB_OPEN )
   END_RUNG wire#w5
   RUNG wire#w1
      Contact( "IO_Valve_Buffer_DB"."AV-65.21".FB_OPEN )
      Coil( "BFT-66".IN_FBAV_CIP_Line )
   END_RUNG
   // the same network as SCL:
   "BFT-66".IN_FBAV_Inload := "AlwaysTRUE" AND "IO_Valve_Buffer_DB"."AV-66.01".FB_OPEN AND ("IO_Valve_Buffer_DB"."AV-66.02".FB_OPEN OR "IO_Valve_Buffer_DB"."AV-66.03".FB_OPEN);
   "BFT-66".IN_FBAV_CIP_Tank := "AlwaysTRUE" AND "IO_Valve_Buffer_DB"."AV-65.21".FB_OPEN AND ("IO_Valve_Buffer_DB"."AV-66.04".FB_OPEN OR "IO_Valve_Buffer_DB"."AV-66.05".FB_OPEN);
   "BFT-66".IN_FBAV_CIP_Line := "AlwaysTRUE" AND "IO_Valve_Buffer_DB"."AV-65.21".FB_OPEN;
END_REGION

REGION Network 15: Comm BFT 65 and BFT 66 to Blending
   RUNG wire#powerrail
      Contact( "AlwaysTRUE" )
      wire#w1
      Contact( "BFT-65".Out_Prod_Req )
      wire#w2
      Coil( "Blend_T-31"."BFT-2 Prod Req" )
   END_RUNG
   RUNG wire#w1
      Contact( "BFT-66".Out_Prod_Req )
   END_RUNG wire#w2
   RUNG wire#w2
      Coil( "Blend_T-40"."BFT-2 Prod Req" )
   END_RUNG
   RUNG wire#w2
      Coil( "Blend_T-41"."BFT-2 Prod Req" )
   END_RUNG
   RUNG wire#w1
      Contact( "BFT-65".Out_Prod_LineOpen )
      wire#w3
      Coil( "Blend_T-31"."BFT-2 Prod Line" )
   END_RUNG
   RUNG wire#w1
      Contact( "BFT-66".Out_Prod_LineOpen )
   END_RUNG wire#w3
   RUNG wire#w3
      Coil( "Blend_T-40"."BFT-2 Prod Line" )
   END_RUNG
   RUNG wire#w3
      Coil( "Blend_T-41"."BFT-2 Prod Line" )
   END_RUNG
   // the same network as SCL:
   "Blend_T-31"."BFT-2 Prod Req" := "AlwaysTRUE" AND ("BFT-65".Out_Prod_Req OR "BFT-66".Out_Prod_Req);
   "Blend_T-40"."BFT-2 Prod Req" := "Blend_T-31"."BFT-2 Prod Req";
   "Blend_T-41"."BFT-2 Prod Req" := "Blend_T-31"."BFT-2 Prod Req";
   "Blend_T-31"."BFT-2 Prod Line" := "AlwaysTRUE" AND ("BFT-65".Out_Prod_LineOpen OR "BFT-66".Out_Prod_LineOpen);
   "Blend_T-40"."BFT-2 Prod Line" := "Blend_T-31"."BFT-2 Prod Line";
   "Blend_T-41"."BFT-2 Prod Line" := "Blend_T-31"."BFT-2 Prod Line";
END_REGION

REGION Network 16: Comm CIP Line 65 & 66
   RUNG wire#powerrail
      Contact( "AlwaysTRUE" )
      wire#w1
      Contact( "BFT-65".Out_CIP_Line_Req )
      wire#w2
      Coil( "Mix_to_CIP".CIP_Request."Buffer Cluster 2"."T65&T66_CIP_LineToPasteur_Request" )
   END_RUNG
   RUNG wire#w1
      Contact( "BFT-66".Out_CIP_Line_Req )
   END_RUNG wire#w2
   RUNG wire#w1
      Contact( "BFT-65".Out_CIP_Line_LineOpen )
      wire#w3
      Coil( "Mix_to_CIP".CIP_Line_OK."Buffer Cluster 2"."T65&T66_CIP_LineToPasteur_LineOK" )
   END_RUNG
   RUNG wire#w1
      Contact( "BFT-66".Out_CIP_Line_LineOpen )
   END_RUNG wire#w3
   // the same network as SCL:
   "Mix_to_CIP".CIP_Request."Buffer Cluster 2"."T65&T66_CIP_LineToPasteur_Request" := "AlwaysTRUE" AND ("BFT-65".Out_CIP_Line_Req OR "BFT-66".Out_CIP_Line_Req);
   "Mix_to_CIP".CIP_Line_OK."Buffer Cluster 2"."T65&T66_CIP_LineToPasteur_LineOK" := "AlwaysTRUE" AND ("BFT-65".Out_CIP_Line_LineOpen OR "BFT-66".Out_CIP_Line_LineOpen);
END_REGION

REGION Network 18: BFT 67
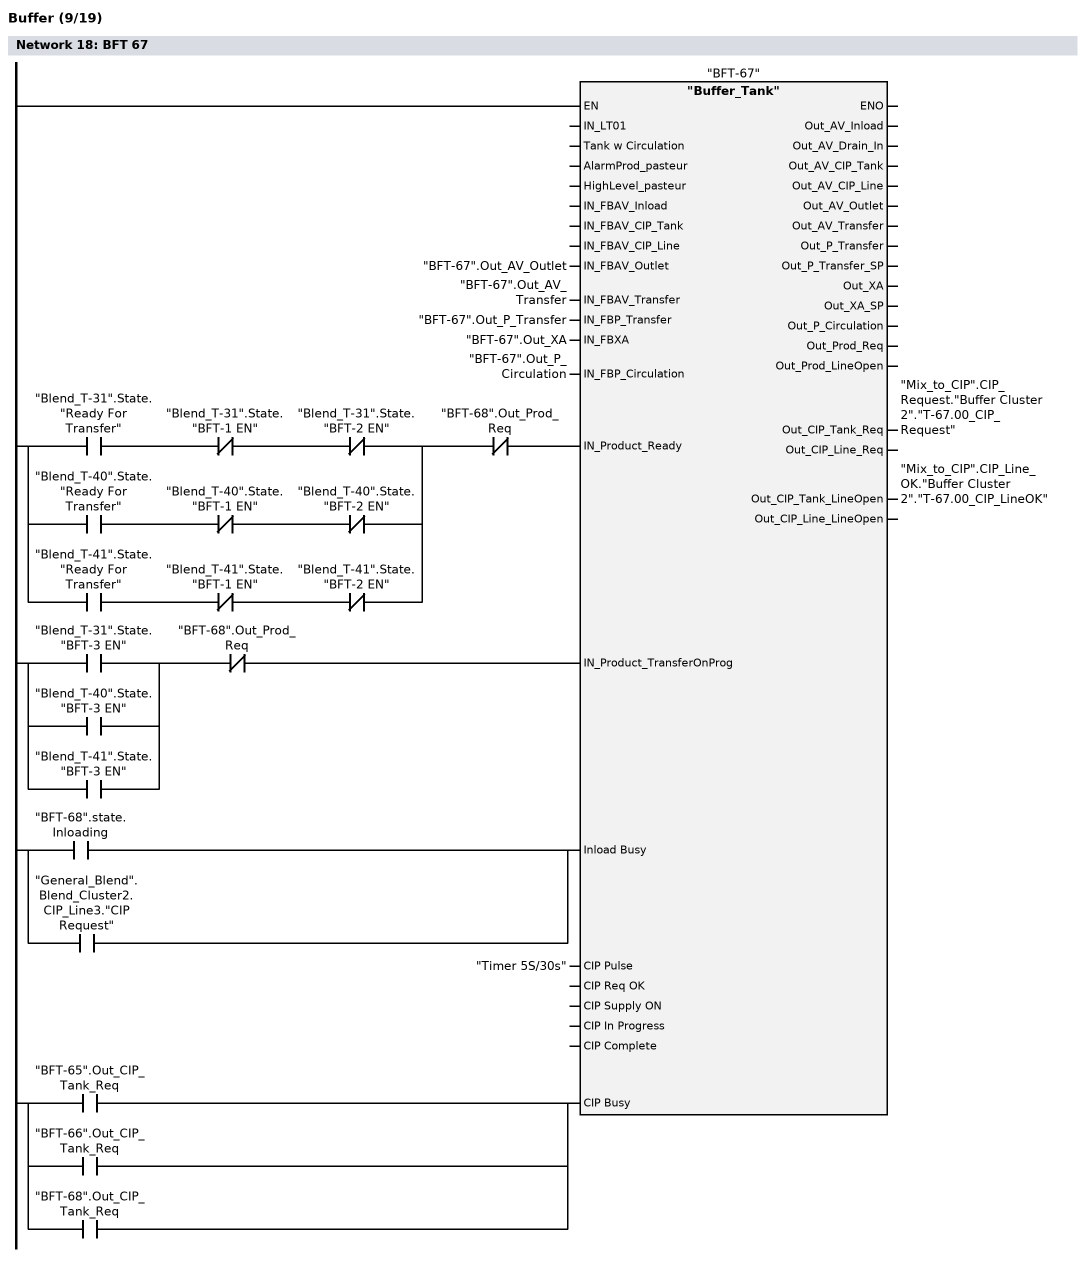
   RUNG wire#powerrail
      "BFT-67"(IN_Product_Ready := wire#w2, IN_Product_TransferOnProg := wire#w4, "Inload Busy" := wire#w5, "CIP Busy" := wire#w6, IN_LT01 :=, "Tank w Circulation" :=, AlarmProd_pasteur :=, HighLevel_pasteur :=, IN_FBAV_Inload :=, IN_FBAV_CIP_Tank :=, IN_FBAV_CIP_Line :=, IN_FBAV_Outlet := "BFT-67".Out_AV_Outlet, IN_FBAV_Transfer := "BFT-67".Out_AV_Transfer, IN_FBP_Transfer := "BFT-67".Out_P_Transfer, IN_FBXA := "BFT-67".Out_XA, IN_FBP_Circulation := "BFT-67".Out_P_Circulation, "CIP Pulse" := "Timer 5S/30s", "CIP Req OK" :=, "CIP Supply ON" :=, "CIP In Progress" :=, "CIP Complete" :=, Out_AV_Inload =>, Out_AV_Drain_In =>, Out_AV_CIP_Tank =>, Out_AV_CIP_Line =>, Out_AV_Outlet =>, Out_AV_Transfer =>, Out_P_Transfer =>, Out_P_Transfer_SP =>, Out_XA =>, Out_XA_SP =>, Out_P_Circulation =>, Out_Prod_Req =>, Out_Prod_LineOpen =>, Out_CIP_Tank_Req => "Mix_to_CIP".CIP_Request."Buffer Cluster 2"."T-67.00_CIP_Request", Out_CIP_Line_Req =>, Out_CIP_Tank_LineOpen => "Mix_to_CIP".CIP_Line_OK."Buffer Cluster 2"."T-67.00_CIP_LineOK", Out_CIP_Line_LineOpen =>)
   END_RUNG
   RUNG wire#powerrail
      Contact( "Blend_T-31".State."Ready For Transfer" )
      I_Contact( "Blend_T-31".State."BFT-1 EN" )
      I_Contact( "Blend_T-31".State."BFT-2 EN" )
      wire#w1
      I_Contact( "BFT-68".Out_Prod_Req )
   END_RUNG wire#w2
   RUNG wire#powerrail
      Contact( "Blend_T-40".State."Ready For Transfer" )
      I_Contact( "Blend_T-40".State."BFT-1 EN" )
      I_Contact( "Blend_T-40".State."BFT-2 EN" )
   END_RUNG wire#w1
   RUNG wire#powerrail
      Contact( "Blend_T-41".State."Ready For Transfer" )
      I_Contact( "Blend_T-41".State."BFT-1 EN" )
      I_Contact( "Blend_T-41".State."BFT-2 EN" )
   END_RUNG wire#w1
   RUNG wire#powerrail
      Contact( "Blend_T-31".State."BFT-3 EN" )
      wire#w3
      I_Contact( "BFT-68".Out_Prod_Req )
   END_RUNG wire#w4
   RUNG wire#powerrail
      Contact( "Blend_T-40".State."BFT-3 EN" )
   END_RUNG wire#w3
   RUNG wire#powerrail
      Contact( "Blend_T-41".State."BFT-3 EN" )
   END_RUNG wire#w3
   RUNG wire#powerrail
      Contact( "BFT-68".state.Inloading )
   END_RUNG wire#w5
   RUNG wire#powerrail
      Contact( "General_Blend".Blend_Cluster2.CIP_Line3."CIP Request" )
   END_RUNG wire#w5
   RUNG wire#powerrail
      Contact( "BFT-65".Out_CIP_Tank_Req )
   END_RUNG wire#w6
   RUNG wire#powerrail
      Contact( "BFT-66".Out_CIP_Tank_Req )
   END_RUNG wire#w6
   RUNG wire#powerrail
      Contact( "BFT-68".Out_CIP_Tank_Req )
   END_RUNG wire#w6
   // the same network as SCL:
   "BFT-67"(IN_FBAV_Outlet := "BFT-67".Out_AV_Outlet,   // "Buffer_Tank"
            IN_FBAV_Transfer := "BFT-67".Out_AV_Transfer,
            IN_FBP_Transfer := "BFT-67".Out_P_Transfer,
            IN_FBXA := "BFT-67".Out_XA,
            IN_FBP_Circulation := "BFT-67".Out_P_Circulation,
            IN_Product_Ready := (("Blend_T-31".State."Ready For Transfer" AND NOT "Blend_T-31".State."BFT-1 EN" AND NOT "Blend_T-31".State."BFT-2 EN") OR ("Blend_T-40".State."Ready For Transfer" AND NOT "Blend_T-40".State."BFT-1 EN" AND NOT "Blend_T-40".State."BFT-2 EN") OR ("Blend_T-41".State."Ready For Transfer" AND NOT "Blend_T-41".State."BFT-1 EN" AND NOT "Blend_T-41".State."BFT-2 EN")) AND NOT "BFT-68".Out_Prod_Req,
            IN_Product_TransferOnProg := ("Blend_T-31".State."BFT-3 EN" OR "Blend_T-40".State."BFT-3 EN" OR "Blend_T-41".State."BFT-3 EN") AND NOT "BFT-68".Out_Prod_Req,
            "Inload Busy" := "BFT-68".state.Inloading OR "General_Blend".Blend_Cluster2.CIP_Line3."CIP Request",
            "CIP Pulse" := "Timer 5S/30s",
            "CIP Busy" := "BFT-65".Out_CIP_Tank_Req OR "BFT-66".Out_CIP_Tank_Req OR "BFT-68".Out_CIP_Tank_Req,
            Out_CIP_Tank_Req => "Mix_to_CIP".CIP_Request."Buffer Cluster 2"."T-67.00_CIP_Request",
            Out_CIP_Tank_LineOpen => "Mix_to_CIP".CIP_Line_OK."Buffer Cluster 2"."T-67.00_CIP_LineOK");
END_REGION

REGION Network 19: BFT 67 Feedback Instrument
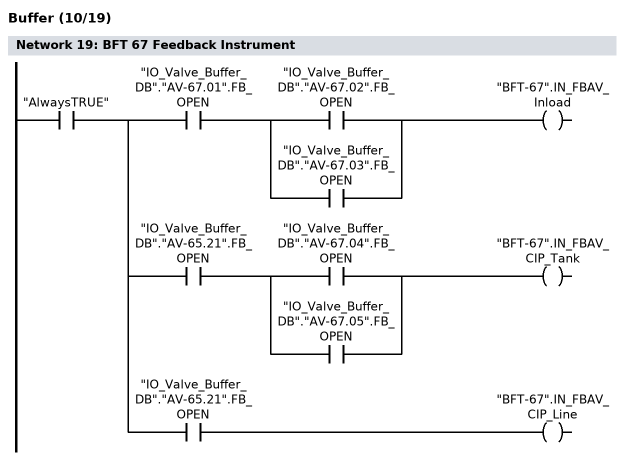
   RUNG wire#powerrail
      Contact( "AlwaysTRUE" )
      wire#w1
      Contact( "IO_Valve_Buffer_DB"."AV-67.01".FB_OPEN )
      wire#w2
      Contact( "IO_Valve_Buffer_DB"."AV-67.02".FB_OPEN )
      wire#w3
      Coil( "BFT-67".IN_FBAV_Inload )
   END_RUNG
   RUNG wire#w2
      Contact( "IO_Valve_Buffer_DB"."AV-67.03".FB_OPEN )
   END_RUNG wire#w3
   RUNG wire#w1
      Contact( "IO_Valve_Buffer_DB"."AV-65.21".FB_OPEN )
      wire#w4
      Contact( "IO_Valve_Buffer_DB"."AV-67.04".FB_OPEN )
      wire#w5
      Coil( "BFT-67".IN_FBAV_CIP_Tank )
   END_RUNG
   RUNG wire#w4
      Contact( "IO_Valve_Buffer_DB"."AV-67.05".FB_OPEN )
   END_RUNG wire#w5
   RUNG wire#w1
      Contact( "IO_Valve_Buffer_DB"."AV-65.21".FB_OPEN )
      Coil( "BFT-67".IN_FBAV_CIP_Line )
   END_RUNG
   // the same network as SCL:
   "BFT-67".IN_FBAV_Inload := "AlwaysTRUE" AND "IO_Valve_Buffer_DB"."AV-67.01".FB_OPEN AND ("IO_Valve_Buffer_DB"."AV-67.02".FB_OPEN OR "IO_Valve_Buffer_DB"."AV-67.03".FB_OPEN);
   "BFT-67".IN_FBAV_CIP_Tank := "AlwaysTRUE" AND "IO_Valve_Buffer_DB"."AV-65.21".FB_OPEN AND ("IO_Valve_Buffer_DB"."AV-67.04".FB_OPEN OR "IO_Valve_Buffer_DB"."AV-67.05".FB_OPEN);
   "BFT-67".IN_FBAV_CIP_Line := "AlwaysTRUE" AND "IO_Valve_Buffer_DB"."AV-65.21".FB_OPEN;
END_REGION

REGION Network 20: BFT 68
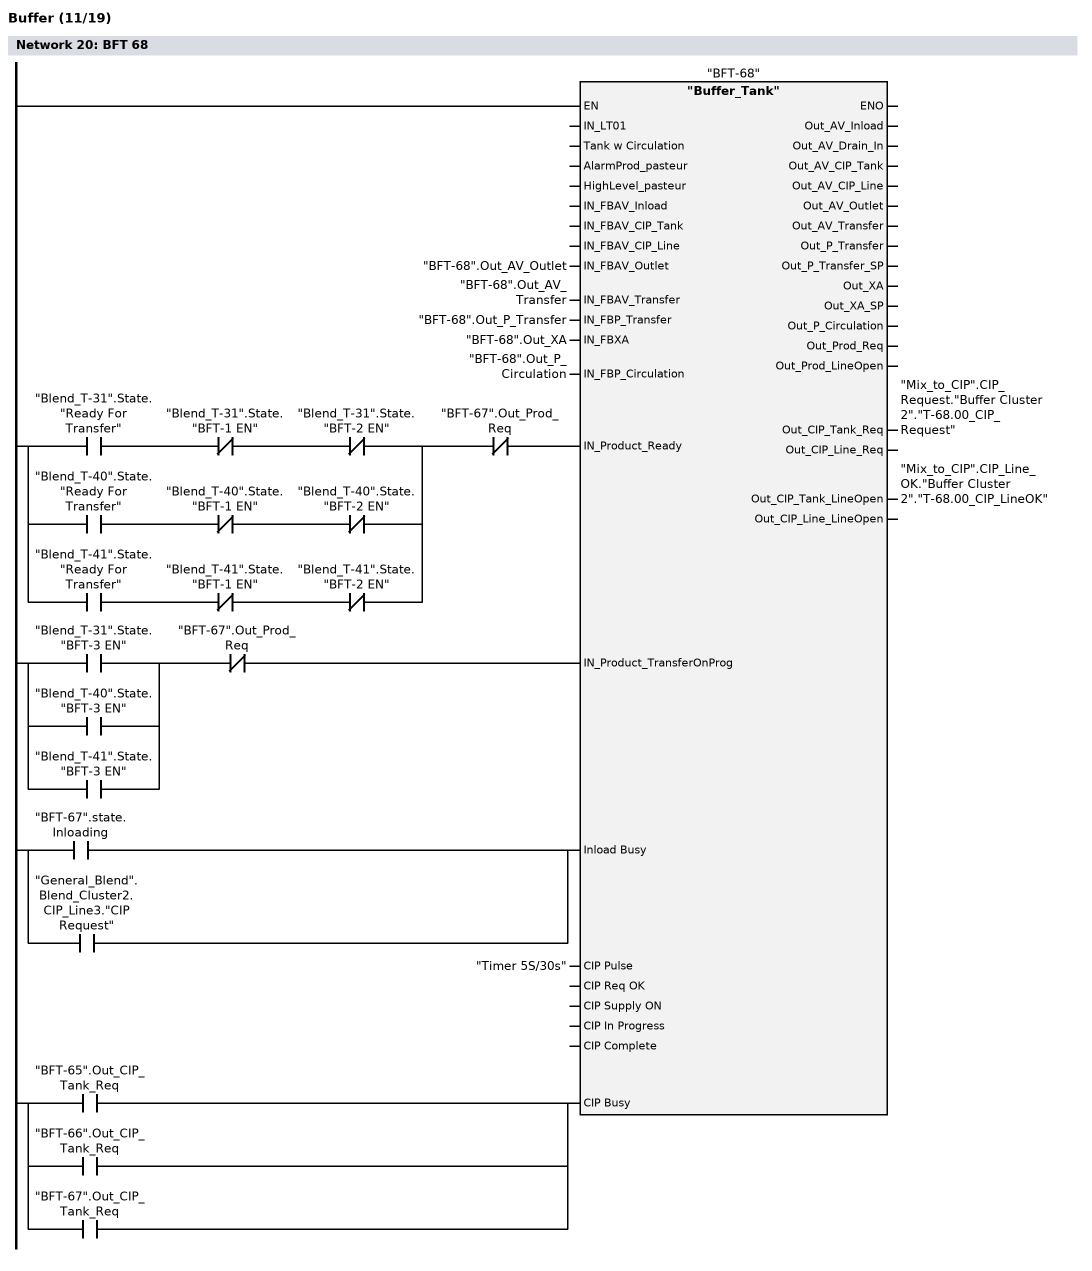
   RUNG wire#powerrail
      "BFT-68"(IN_Product_Ready := wire#w2, IN_Product_TransferOnProg := wire#w4, "Inload Busy" := wire#w5, "CIP Busy" := wire#w6, IN_LT01 :=, "Tank w Circulation" :=, AlarmProd_pasteur :=, HighLevel_pasteur :=, IN_FBAV_Inload :=, IN_FBAV_CIP_Tank :=, IN_FBAV_CIP_Line :=, IN_FBAV_Outlet := "BFT-68".Out_AV_Outlet, IN_FBAV_Transfer := "BFT-68".Out_AV_Transfer, IN_FBP_Transfer := "BFT-68".Out_P_Transfer, IN_FBXA := "BFT-68".Out_XA, IN_FBP_Circulation := "BFT-68".Out_P_Circulation, "CIP Pulse" := "Timer 5S/30s", "CIP Req OK" :=, "CIP Supply ON" :=, "CIP In Progress" :=, "CIP Complete" :=, Out_AV_Inload =>, Out_AV_Drain_In =>, Out_AV_CIP_Tank =>, Out_AV_CIP_Line =>, Out_AV_Outlet =>, Out_AV_Transfer =>, Out_P_Transfer =>, Out_P_Transfer_SP =>, Out_XA =>, Out_XA_SP =>, Out_P_Circulation =>, Out_Prod_Req =>, Out_Prod_LineOpen =>, Out_CIP_Tank_Req => "Mix_to_CIP".CIP_Request."Buffer Cluster 2"."T-68.00_CIP_Request", Out_CIP_Line_Req =>, Out_CIP_Tank_LineOpen => "Mix_to_CIP".CIP_Line_OK."Buffer Cluster 2"."T-68.00_CIP_LineOK", Out_CIP_Line_LineOpen =>)
   END_RUNG
   RUNG wire#powerrail
      Contact( "Blend_T-31".State."Ready For Transfer" )
      I_Contact( "Blend_T-31".State."BFT-1 EN" )
      I_Contact( "Blend_T-31".State."BFT-2 EN" )
      wire#w1
      I_Contact( "BFT-67".Out_Prod_Req )
   END_RUNG wire#w2
   RUNG wire#powerrail
      Contact( "Blend_T-40".State."Ready For Transfer" )
      I_Contact( "Blend_T-40".State."BFT-1 EN" )
      I_Contact( "Blend_T-40".State."BFT-2 EN" )
   END_RUNG wire#w1
   RUNG wire#powerrail
      Contact( "Blend_T-41".State."Ready For Transfer" )
      I_Contact( "Blend_T-41".State."BFT-1 EN" )
      I_Contact( "Blend_T-41".State."BFT-2 EN" )
   END_RUNG wire#w1
   RUNG wire#powerrail
      Contact( "Blend_T-31".State."BFT-3 EN" )
      wire#w3
      I_Contact( "BFT-67".Out_Prod_Req )
   END_RUNG wire#w4
   RUNG wire#powerrail
      Contact( "Blend_T-40".State."BFT-3 EN" )
   END_RUNG wire#w3
   RUNG wire#powerrail
      Contact( "Blend_T-41".State."BFT-3 EN" )
   END_RUNG wire#w3
   RUNG wire#powerrail
      Contact( "BFT-67".state.Inloading )
   END_RUNG wire#w5
   RUNG wire#powerrail
      Contact( "General_Blend".Blend_Cluster2.CIP_Line3."CIP Request" )
   END_RUNG wire#w5
   RUNG wire#powerrail
      Contact( "BFT-65".Out_CIP_Tank_Req )
   END_RUNG wire#w6
   RUNG wire#powerrail
      Contact( "BFT-66".Out_CIP_Tank_Req )
   END_RUNG wire#w6
   RUNG wire#powerrail
      Contact( "BFT-67".Out_CIP_Tank_Req )
   END_RUNG wire#w6
   // the same network as SCL:
   "BFT-68"(IN_FBAV_Outlet := "BFT-68".Out_AV_Outlet,   // "Buffer_Tank"
            IN_FBAV_Transfer := "BFT-68".Out_AV_Transfer,
            IN_FBP_Transfer := "BFT-68".Out_P_Transfer,
            IN_FBXA := "BFT-68".Out_XA,
            IN_FBP_Circulation := "BFT-68".Out_P_Circulation,
            IN_Product_Ready := (("Blend_T-31".State."Ready For Transfer" AND NOT "Blend_T-31".State."BFT-1 EN" AND NOT "Blend_T-31".State."BFT-2 EN") OR ("Blend_T-40".State."Ready For Transfer" AND NOT "Blend_T-40".State."BFT-1 EN" AND NOT "Blend_T-40".State."BFT-2 EN") OR ("Blend_T-41".State."Ready For Transfer" AND NOT "Blend_T-41".State."BFT-1 EN" AND NOT "Blend_T-41".State."BFT-2 EN")) AND NOT "BFT-67".Out_Prod_Req,
            IN_Product_TransferOnProg := ("Blend_T-31".State."BFT-3 EN" OR "Blend_T-40".State."BFT-3 EN" OR "Blend_T-41".State."BFT-3 EN") AND NOT "BFT-67".Out_Prod_Req,
            "Inload Busy" := "BFT-67".state.Inloading OR "General_Blend".Blend_Cluster2.CIP_Line3."CIP Request",
            "CIP Pulse" := "Timer 5S/30s",
            "CIP Busy" := "BFT-65".Out_CIP_Tank_Req OR "BFT-66".Out_CIP_Tank_Req OR "BFT-67".Out_CIP_Tank_Req,
            Out_CIP_Tank_Req => "Mix_to_CIP".CIP_Request."Buffer Cluster 2"."T-68.00_CIP_Request",
            Out_CIP_Tank_LineOpen => "Mix_to_CIP".CIP_Line_OK."Buffer Cluster 2"."T-68.00_CIP_LineOK");
END_REGION

REGION Network 21: BFT 68 Feedback Instrument
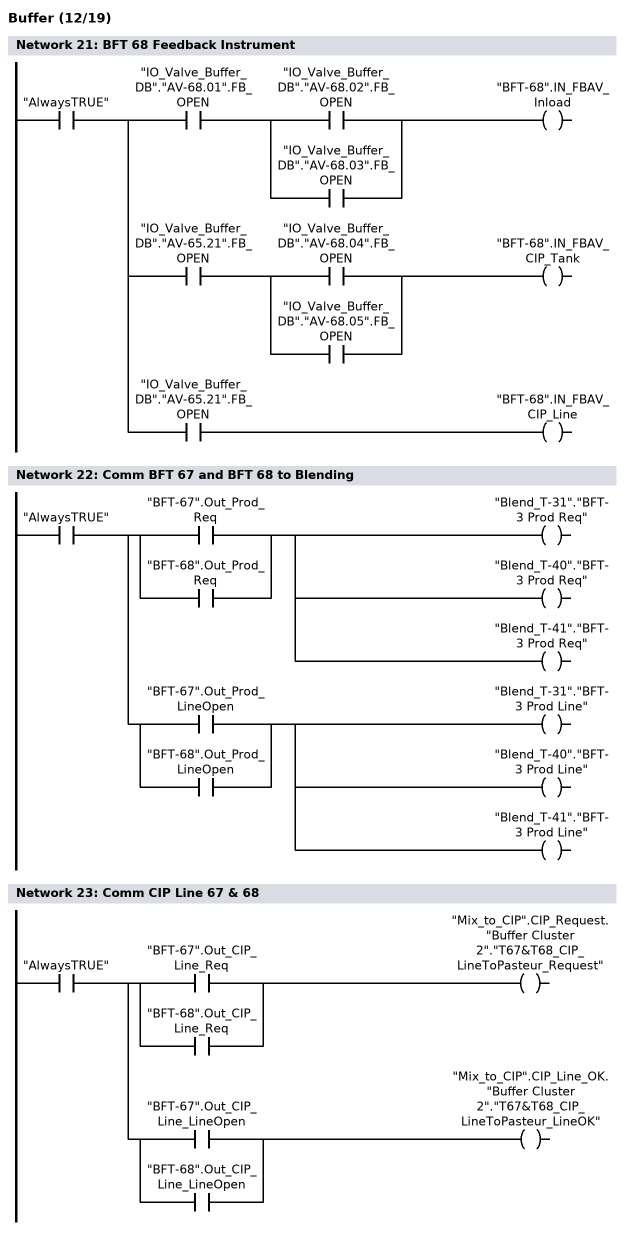
   RUNG wire#powerrail
      Contact( "AlwaysTRUE" )
      wire#w1
      Contact( "IO_Valve_Buffer_DB"."AV-68.01".FB_OPEN )
      wire#w2
      Contact( "IO_Valve_Buffer_DB"."AV-68.02".FB_OPEN )
      wire#w3
      Coil( "BFT-68".IN_FBAV_Inload )
   END_RUNG
   RUNG wire#w2
      Contact( "IO_Valve_Buffer_DB"."AV-68.03".FB_OPEN )
   END_RUNG wire#w3
   RUNG wire#w1
      Contact( "IO_Valve_Buffer_DB"."AV-65.21".FB_OPEN )
      wire#w4
      Contact( "IO_Valve_Buffer_DB"."AV-68.04".FB_OPEN )
      wire#w5
      Coil( "BFT-68".IN_FBAV_CIP_Tank )
   END_RUNG
   RUNG wire#w4
      Contact( "IO_Valve_Buffer_DB"."AV-68.05".FB_OPEN )
   END_RUNG wire#w5
   RUNG wire#w1
      Contact( "IO_Valve_Buffer_DB"."AV-65.21".FB_OPEN )
      Coil( "BFT-68".IN_FBAV_CIP_Line )
   END_RUNG
   // the same network as SCL:
   "BFT-68".IN_FBAV_Inload := "AlwaysTRUE" AND "IO_Valve_Buffer_DB"."AV-68.01".FB_OPEN AND ("IO_Valve_Buffer_DB"."AV-68.02".FB_OPEN OR "IO_Valve_Buffer_DB"."AV-68.03".FB_OPEN);
   "BFT-68".IN_FBAV_CIP_Tank := "AlwaysTRUE" AND "IO_Valve_Buffer_DB"."AV-65.21".FB_OPEN AND ("IO_Valve_Buffer_DB"."AV-68.04".FB_OPEN OR "IO_Valve_Buffer_DB"."AV-68.05".FB_OPEN);
   "BFT-68".IN_FBAV_CIP_Line := "AlwaysTRUE" AND "IO_Valve_Buffer_DB"."AV-65.21".FB_OPEN;
END_REGION

REGION Network 22: Comm BFT 67 and BFT 68 to Blending
   RUNG wire#powerrail
      Contact( "AlwaysTRUE" )
      wire#w1
      Contact( "BFT-67".Out_Prod_Req )
      wire#w2
      Coil( "Blend_T-31"."BFT-3 Prod Req" )
   END_RUNG
   RUNG wire#w1
      Contact( "BFT-68".Out_Prod_Req )
   END_RUNG wire#w2
   RUNG wire#w2
      Coil( "Blend_T-40"."BFT-3 Prod Req" )
   END_RUNG
   RUNG wire#w2
      Coil( "Blend_T-41"."BFT-3 Prod Req" )
   END_RUNG
   RUNG wire#w1
      Contact( "BFT-67".Out_Prod_LineOpen )
      wire#w3
      Coil( "Blend_T-31"."BFT-3 Prod Line" )
   END_RUNG
   RUNG wire#w1
      Contact( "BFT-68".Out_Prod_LineOpen )
   END_RUNG wire#w3
   RUNG wire#w3
      Coil( "Blend_T-40"."BFT-3 Prod Line" )
   END_RUNG
   RUNG wire#w3
      Coil( "Blend_T-41"."BFT-3 Prod Line" )
   END_RUNG
   // the same network as SCL:
   "Blend_T-31"."BFT-3 Prod Req" := "AlwaysTRUE" AND ("BFT-67".Out_Prod_Req OR "BFT-68".Out_Prod_Req);
   "Blend_T-40"."BFT-3 Prod Req" := "Blend_T-31"."BFT-3 Prod Req";
   "Blend_T-41"."BFT-3 Prod Req" := "Blend_T-31"."BFT-3 Prod Req";
   "Blend_T-31"."BFT-3 Prod Line" := "AlwaysTRUE" AND ("BFT-67".Out_Prod_LineOpen OR "BFT-68".Out_Prod_LineOpen);
   "Blend_T-40"."BFT-3 Prod Line" := "Blend_T-31"."BFT-3 Prod Line";
   "Blend_T-41"."BFT-3 Prod Line" := "Blend_T-31"."BFT-3 Prod Line";
END_REGION

REGION Network 23: Comm CIP Line 67 & 68
   RUNG wire#powerrail
      Contact( "AlwaysTRUE" )
      wire#w1
      Contact( "BFT-67".Out_CIP_Line_Req )
      wire#w2
      Coil( "Mix_to_CIP".CIP_Request."Buffer Cluster 2"."T67&T68_CIP_LineToPasteur_Request" )
   END_RUNG
   RUNG wire#w1
      Contact( "BFT-68".Out_CIP_Line_Req )
   END_RUNG wire#w2
   RUNG wire#w1
      Contact( "BFT-67".Out_CIP_Line_LineOpen )
      wire#w3
      Coil( "Mix_to_CIP".CIP_Line_OK."Buffer Cluster 2"."T67&T68_CIP_LineToPasteur_LineOK" )
   END_RUNG
   RUNG wire#w1
      Contact( "BFT-68".Out_CIP_Line_LineOpen )
   END_RUNG wire#w3
   // the same network as SCL:
   "Mix_to_CIP".CIP_Request."Buffer Cluster 2"."T67&T68_CIP_LineToPasteur_Request" := "AlwaysTRUE" AND ("BFT-67".Out_CIP_Line_Req OR "BFT-68".Out_CIP_Line_Req);
   "Mix_to_CIP".CIP_Line_OK."Buffer Cluster 2"."T67&T68_CIP_LineToPasteur_LineOK" := "AlwaysTRUE" AND ("BFT-67".Out_CIP_Line_LineOpen OR "BFT-68".Out_CIP_Line_LineOpen);
END_REGION

REGION Network 25: Comm CIP to BFT 61 Rework 32
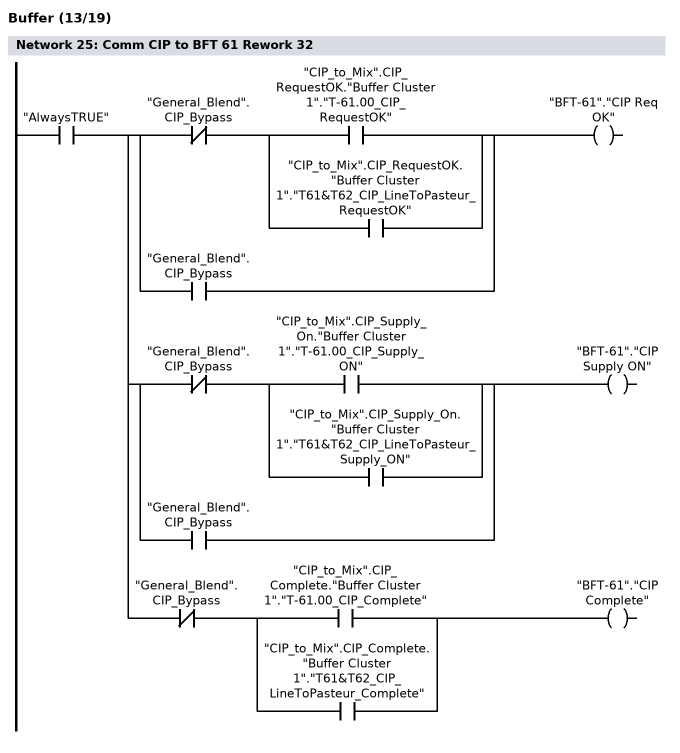
   RUNG wire#powerrail
      Contact( "AlwaysTRUE" )
      wire#w1
      I_Contact( "General_Blend".CIP_Bypass )
      wire#w2
      Contact( "CIP_to_Mix".CIP_RequestOK."Buffer Cluster 1"."T-61.00_CIP_RequestOK" )
      wire#w3
      Coil( "BFT-61"."CIP Req OK" )
   END_RUNG
   RUNG wire#w2
      Contact( "CIP_to_Mix".CIP_RequestOK."Buffer Cluster 1"."T61&T62_CIP_LineToPasteur_RequestOK" )
   END_RUNG wire#w3
   RUNG wire#w1
      Contact( "General_Blend".CIP_Bypass )
   END_RUNG wire#w3
   RUNG wire#w1
      I_Contact( "General_Blend".CIP_Bypass )
      wire#w4
      Contact( "CIP_to_Mix".CIP_Supply_On."Buffer Cluster 1"."T-61.00_CIP_Supply_ON" )
      wire#w5
      Coil( "BFT-61"."CIP Supply ON" )
   END_RUNG
   RUNG wire#w4
      Contact( "CIP_to_Mix".CIP_Supply_On."Buffer Cluster 1"."T61&T62_CIP_LineToPasteur_Supply_ON" )
   END_RUNG wire#w5
   RUNG wire#w1
      Contact( "General_Blend".CIP_Bypass )
   END_RUNG wire#w5
   RUNG wire#w1
      I_Contact( "General_Blend".CIP_Bypass )
      wire#w6
      Contact( "CIP_to_Mix".CIP_Complete."Buffer Cluster 1"."T-61.00_CIP_Complete" )
      wire#w7
      Coil( "BFT-61"."CIP Complete" )
   END_RUNG
   RUNG wire#w6
      Contact( "CIP_to_Mix".CIP_Complete."Buffer Cluster 1"."T61&T62_CIP_LineToPasteur_Complete" )
   END_RUNG wire#w7
   // the same network as SCL:
   "BFT-61"."CIP Req OK" := "AlwaysTRUE" AND ((NOT "General_Blend".CIP_Bypass AND ("CIP_to_Mix".CIP_RequestOK."Buffer Cluster 1"."T-61.00_CIP_RequestOK" OR "CIP_to_Mix".CIP_RequestOK."Buffer Cluster 1"."T61&T62_CIP_LineToPasteur_RequestOK")) OR "General_Blend".CIP_Bypass);
   "BFT-61"."CIP Supply ON" := "AlwaysTRUE" AND ((NOT "General_Blend".CIP_Bypass AND ("CIP_to_Mix".CIP_Supply_On."Buffer Cluster 1"."T-61.00_CIP_Supply_ON" OR "CIP_to_Mix".CIP_Supply_On."Buffer Cluster 1"."T61&T62_CIP_LineToPasteur_Supply_ON")) OR "General_Blend".CIP_Bypass);
   "BFT-61"."CIP Complete" := "AlwaysTRUE" AND NOT "General_Blend".CIP_Bypass AND ("CIP_to_Mix".CIP_Complete."Buffer Cluster 1"."T-61.00_CIP_Complete" OR "CIP_to_Mix".CIP_Complete."Buffer Cluster 1"."T61&T62_CIP_LineToPasteur_Complete");
END_REGION

REGION Network 26: Comm CIP to BFT 64 Rework 22
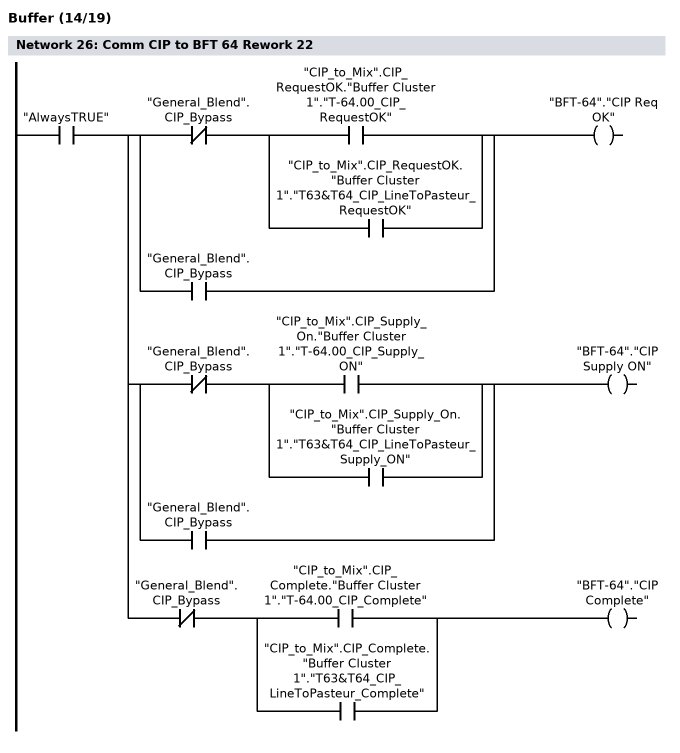
   RUNG wire#powerrail
      Contact( "AlwaysTRUE" )
      wire#w1
      I_Contact( "General_Blend".CIP_Bypass )
      wire#w2
      Contact( "CIP_to_Mix".CIP_RequestOK."Buffer Cluster 1"."T-64.00_CIP_RequestOK" )
      wire#w3
      Coil( "BFT-64"."CIP Req OK" )
   END_RUNG
   RUNG wire#w2
      Contact( "CIP_to_Mix".CIP_RequestOK."Buffer Cluster 1"."T63&T64_CIP_LineToPasteur_RequestOK" )
   END_RUNG wire#w3
   RUNG wire#w1
      Contact( "General_Blend".CIP_Bypass )
   END_RUNG wire#w3
   RUNG wire#w1
      I_Contact( "General_Blend".CIP_Bypass )
      wire#w4
      Contact( "CIP_to_Mix".CIP_Supply_On."Buffer Cluster 1"."T-64.00_CIP_Supply_ON" )
      wire#w5
      Coil( "BFT-64"."CIP Supply ON" )
   END_RUNG
   RUNG wire#w4
      Contact( "CIP_to_Mix".CIP_Supply_On."Buffer Cluster 1"."T63&T64_CIP_LineToPasteur_Supply_ON" )
   END_RUNG wire#w5
   RUNG wire#w1
      Contact( "General_Blend".CIP_Bypass )
   END_RUNG wire#w5
   RUNG wire#w1
      I_Contact( "General_Blend".CIP_Bypass )
      wire#w6
      Contact( "CIP_to_Mix".CIP_Complete."Buffer Cluster 1"."T-64.00_CIP_Complete" )
      wire#w7
      Coil( "BFT-64"."CIP Complete" )
   END_RUNG
   RUNG wire#w6
      Contact( "CIP_to_Mix".CIP_Complete."Buffer Cluster 1"."T63&T64_CIP_LineToPasteur_Complete" )
   END_RUNG wire#w7
   // the same network as SCL:
   "BFT-64"."CIP Req OK" := "AlwaysTRUE" AND ((NOT "General_Blend".CIP_Bypass AND ("CIP_to_Mix".CIP_RequestOK."Buffer Cluster 1"."T-64.00_CIP_RequestOK" OR "CIP_to_Mix".CIP_RequestOK."Buffer Cluster 1"."T63&T64_CIP_LineToPasteur_RequestOK")) OR "General_Blend".CIP_Bypass);
   "BFT-64"."CIP Supply ON" := "AlwaysTRUE" AND ((NOT "General_Blend".CIP_Bypass AND ("CIP_to_Mix".CIP_Supply_On."Buffer Cluster 1"."T-64.00_CIP_Supply_ON" OR "CIP_to_Mix".CIP_Supply_On."Buffer Cluster 1"."T63&T64_CIP_LineToPasteur_Supply_ON")) OR "General_Blend".CIP_Bypass);
   "BFT-64"."CIP Complete" := "AlwaysTRUE" AND NOT "General_Blend".CIP_Bypass AND ("CIP_to_Mix".CIP_Complete."Buffer Cluster 1"."T-64.00_CIP_Complete" OR "CIP_to_Mix".CIP_Complete."Buffer Cluster 1"."T63&T64_CIP_LineToPasteur_Complete");
END_REGION

REGION Network 27: Comm CIP to BFT 65
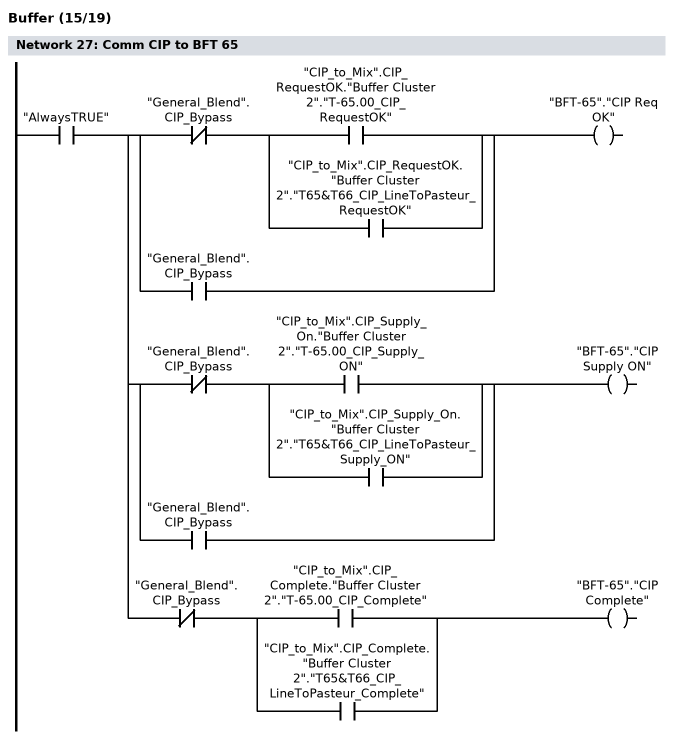
   RUNG wire#powerrail
      Contact( "AlwaysTRUE" )
      wire#w1
      I_Contact( "General_Blend".CIP_Bypass )
      wire#w2
      Contact( "CIP_to_Mix".CIP_RequestOK."Buffer Cluster 2"."T-65.00_CIP_RequestOK" )
      wire#w3
      Coil( "BFT-65"."CIP Req OK" )
   END_RUNG
   RUNG wire#w2
      Contact( "CIP_to_Mix".CIP_RequestOK."Buffer Cluster 2"."T65&T66_CIP_LineToPasteur_RequestOK" )
   END_RUNG wire#w3
   RUNG wire#w1
      Contact( "General_Blend".CIP_Bypass )
   END_RUNG wire#w3
   RUNG wire#w1
      I_Contact( "General_Blend".CIP_Bypass )
      wire#w4
      Contact( "CIP_to_Mix".CIP_Supply_On."Buffer Cluster 2"."T-65.00_CIP_Supply_ON" )
      wire#w5
      Coil( "BFT-65"."CIP Supply ON" )
   END_RUNG
   RUNG wire#w4
      Contact( "CIP_to_Mix".CIP_Supply_On."Buffer Cluster 2"."T65&T66_CIP_LineToPasteur_Supply_ON" )
   END_RUNG wire#w5
   RUNG wire#w1
      Contact( "General_Blend".CIP_Bypass )
   END_RUNG wire#w5
   RUNG wire#w1
      I_Contact( "General_Blend".CIP_Bypass )
      wire#w6
      Contact( "CIP_to_Mix".CIP_Complete."Buffer Cluster 2"."T-65.00_CIP_Complete" )
      wire#w7
      Coil( "BFT-65"."CIP Complete" )
   END_RUNG
   RUNG wire#w6
      Contact( "CIP_to_Mix".CIP_Complete."Buffer Cluster 2"."T65&T66_CIP_LineToPasteur_Complete" )
   END_RUNG wire#w7
   // the same network as SCL:
   "BFT-65"."CIP Req OK" := "AlwaysTRUE" AND ((NOT "General_Blend".CIP_Bypass AND ("CIP_to_Mix".CIP_RequestOK."Buffer Cluster 2"."T-65.00_CIP_RequestOK" OR "CIP_to_Mix".CIP_RequestOK."Buffer Cluster 2"."T65&T66_CIP_LineToPasteur_RequestOK")) OR "General_Blend".CIP_Bypass);
   "BFT-65"."CIP Supply ON" := "AlwaysTRUE" AND ((NOT "General_Blend".CIP_Bypass AND ("CIP_to_Mix".CIP_Supply_On."Buffer Cluster 2"."T-65.00_CIP_Supply_ON" OR "CIP_to_Mix".CIP_Supply_On."Buffer Cluster 2"."T65&T66_CIP_LineToPasteur_Supply_ON")) OR "General_Blend".CIP_Bypass);
   "BFT-65"."CIP Complete" := "AlwaysTRUE" AND NOT "General_Blend".CIP_Bypass AND ("CIP_to_Mix".CIP_Complete."Buffer Cluster 2"."T-65.00_CIP_Complete" OR "CIP_to_Mix".CIP_Complete."Buffer Cluster 2"."T65&T66_CIP_LineToPasteur_Complete");
END_REGION

REGION Network 28: Comm CIP to BFT 66
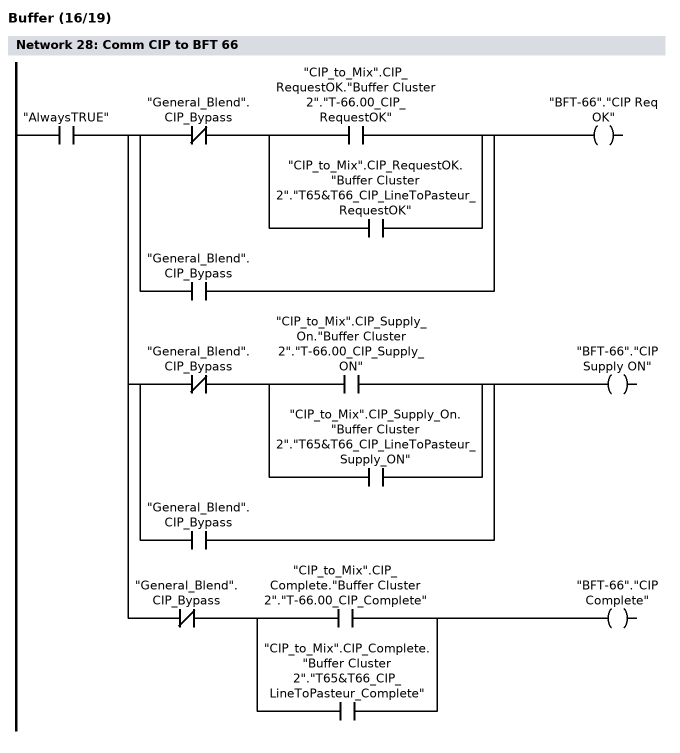
   RUNG wire#powerrail
      Contact( "AlwaysTRUE" )
      wire#w1
      I_Contact( "General_Blend".CIP_Bypass )
      wire#w2
      Contact( "CIP_to_Mix".CIP_RequestOK."Buffer Cluster 2"."T-66.00_CIP_RequestOK" )
      wire#w3
      Coil( "BFT-66"."CIP Req OK" )
   END_RUNG
   RUNG wire#w2
      Contact( "CIP_to_Mix".CIP_RequestOK."Buffer Cluster 2"."T65&T66_CIP_LineToPasteur_RequestOK" )
   END_RUNG wire#w3
   RUNG wire#w1
      Contact( "General_Blend".CIP_Bypass )
   END_RUNG wire#w3
   RUNG wire#w1
      I_Contact( "General_Blend".CIP_Bypass )
      wire#w4
      Contact( "CIP_to_Mix".CIP_Supply_On."Buffer Cluster 2"."T-66.00_CIP_Supply_ON" )
      wire#w5
      Coil( "BFT-66"."CIP Supply ON" )
   END_RUNG
   RUNG wire#w4
      Contact( "CIP_to_Mix".CIP_Supply_On."Buffer Cluster 2"."T65&T66_CIP_LineToPasteur_Supply_ON" )
   END_RUNG wire#w5
   RUNG wire#w1
      Contact( "General_Blend".CIP_Bypass )
   END_RUNG wire#w5
   RUNG wire#w1
      I_Contact( "General_Blend".CIP_Bypass )
      wire#w6
      Contact( "CIP_to_Mix".CIP_Complete."Buffer Cluster 2"."T-66.00_CIP_Complete" )
      wire#w7
      Coil( "BFT-66"."CIP Complete" )
   END_RUNG
   RUNG wire#w6
      Contact( "CIP_to_Mix".CIP_Complete."Buffer Cluster 2"."T65&T66_CIP_LineToPasteur_Complete" )
   END_RUNG wire#w7
   // the same network as SCL:
   "BFT-66"."CIP Req OK" := "AlwaysTRUE" AND ((NOT "General_Blend".CIP_Bypass AND ("CIP_to_Mix".CIP_RequestOK."Buffer Cluster 2"."T-66.00_CIP_RequestOK" OR "CIP_to_Mix".CIP_RequestOK."Buffer Cluster 2"."T65&T66_CIP_LineToPasteur_RequestOK")) OR "General_Blend".CIP_Bypass);
   "BFT-66"."CIP Supply ON" := "AlwaysTRUE" AND ((NOT "General_Blend".CIP_Bypass AND ("CIP_to_Mix".CIP_Supply_On."Buffer Cluster 2"."T-66.00_CIP_Supply_ON" OR "CIP_to_Mix".CIP_Supply_On."Buffer Cluster 2"."T65&T66_CIP_LineToPasteur_Supply_ON")) OR "General_Blend".CIP_Bypass);
   "BFT-66"."CIP Complete" := "AlwaysTRUE" AND NOT "General_Blend".CIP_Bypass AND ("CIP_to_Mix".CIP_Complete."Buffer Cluster 2"."T-66.00_CIP_Complete" OR "CIP_to_Mix".CIP_Complete."Buffer Cluster 2"."T65&T66_CIP_LineToPasteur_Complete");
END_REGION

REGION Network 29: Comm CIP to BFT 67
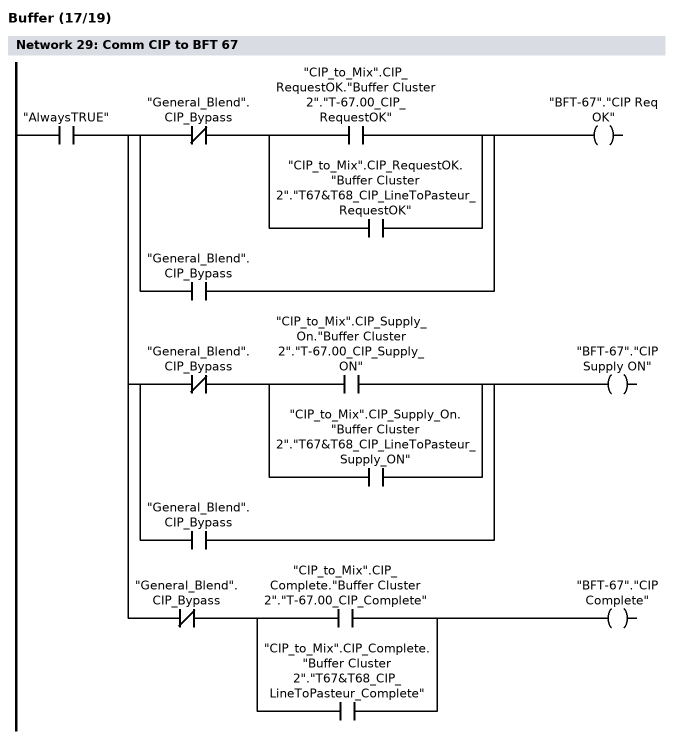
   RUNG wire#powerrail
      Contact( "AlwaysTRUE" )
      wire#w1
      I_Contact( "General_Blend".CIP_Bypass )
      wire#w2
      Contact( "CIP_to_Mix".CIP_RequestOK."Buffer Cluster 2"."T-67.00_CIP_RequestOK" )
      wire#w3
      Coil( "BFT-67"."CIP Req OK" )
   END_RUNG
   RUNG wire#w2
      Contact( "CIP_to_Mix".CIP_RequestOK."Buffer Cluster 2"."T67&T68_CIP_LineToPasteur_RequestOK" )
   END_RUNG wire#w3
   RUNG wire#w1
      Contact( "General_Blend".CIP_Bypass )
   END_RUNG wire#w3
   RUNG wire#w1
      I_Contact( "General_Blend".CIP_Bypass )
      wire#w4
      Contact( "CIP_to_Mix".CIP_Supply_On."Buffer Cluster 2"."T-67.00_CIP_Supply_ON" )
      wire#w5
      Coil( "BFT-67"."CIP Supply ON" )
   END_RUNG
   RUNG wire#w4
      Contact( "CIP_to_Mix".CIP_Supply_On."Buffer Cluster 2"."T67&T68_CIP_LineToPasteur_Supply_ON" )
   END_RUNG wire#w5
   RUNG wire#w1
      Contact( "General_Blend".CIP_Bypass )
   END_RUNG wire#w5
   RUNG wire#w1
      I_Contact( "General_Blend".CIP_Bypass )
      wire#w6
      Contact( "CIP_to_Mix".CIP_Complete."Buffer Cluster 2"."T-67.00_CIP_Complete" )
      wire#w7
      Coil( "BFT-67"."CIP Complete" )
   END_RUNG
   RUNG wire#w6
      Contact( "CIP_to_Mix".CIP_Complete."Buffer Cluster 2"."T67&T68_CIP_LineToPasteur_Complete" )
   END_RUNG wire#w7
   // the same network as SCL:
   "BFT-67"."CIP Req OK" := "AlwaysTRUE" AND ((NOT "General_Blend".CIP_Bypass AND ("CIP_to_Mix".CIP_RequestOK."Buffer Cluster 2"."T-67.00_CIP_RequestOK" OR "CIP_to_Mix".CIP_RequestOK."Buffer Cluster 2"."T67&T68_CIP_LineToPasteur_RequestOK")) OR "General_Blend".CIP_Bypass);
   "BFT-67"."CIP Supply ON" := "AlwaysTRUE" AND ((NOT "General_Blend".CIP_Bypass AND ("CIP_to_Mix".CIP_Supply_On."Buffer Cluster 2"."T-67.00_CIP_Supply_ON" OR "CIP_to_Mix".CIP_Supply_On."Buffer Cluster 2"."T67&T68_CIP_LineToPasteur_Supply_ON")) OR "General_Blend".CIP_Bypass);
   "BFT-67"."CIP Complete" := "AlwaysTRUE" AND NOT "General_Blend".CIP_Bypass AND ("CIP_to_Mix".CIP_Complete."Buffer Cluster 2"."T-67.00_CIP_Complete" OR "CIP_to_Mix".CIP_Complete."Buffer Cluster 2"."T67&T68_CIP_LineToPasteur_Complete");
END_REGION

REGION Network 30: Comm CIP to BFT 68
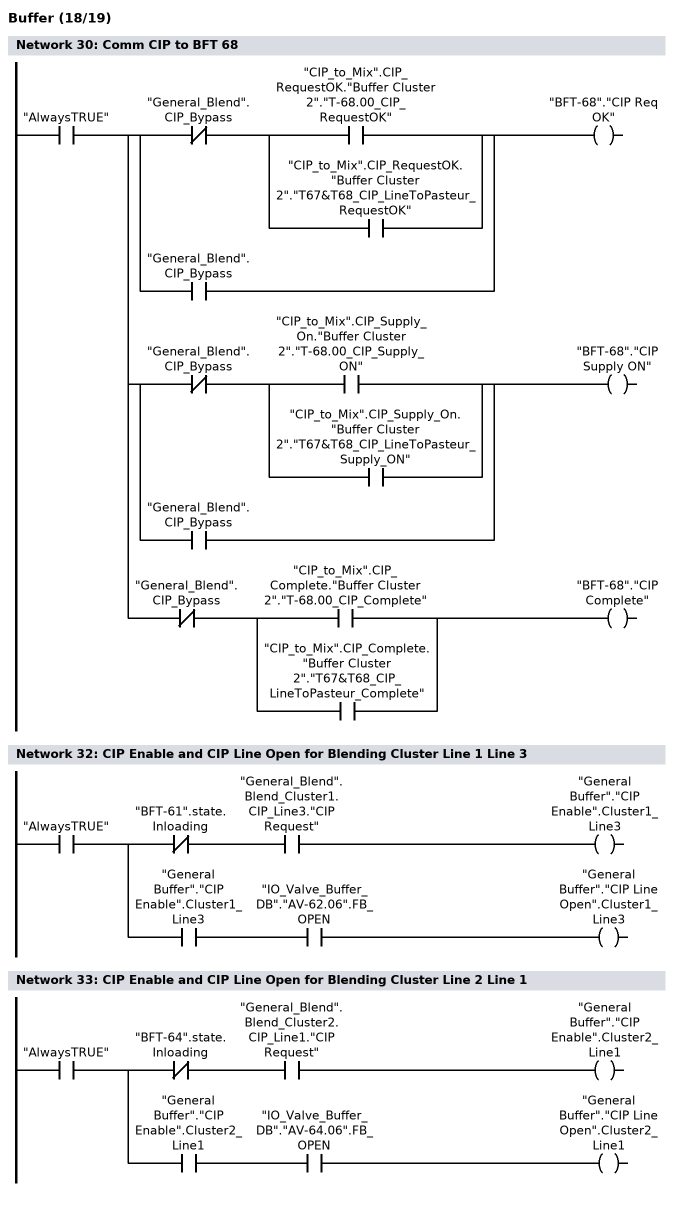
   RUNG wire#powerrail
      Contact( "AlwaysTRUE" )
      wire#w1
      I_Contact( "General_Blend".CIP_Bypass )
      wire#w2
      Contact( "CIP_to_Mix".CIP_RequestOK."Buffer Cluster 2"."T-68.00_CIP_RequestOK" )
      wire#w3
      Coil( "BFT-68"."CIP Req OK" )
   END_RUNG
   RUNG wire#w2
      Contact( "CIP_to_Mix".CIP_RequestOK."Buffer Cluster 2"."T67&T68_CIP_LineToPasteur_RequestOK" )
   END_RUNG wire#w3
   RUNG wire#w1
      Contact( "General_Blend".CIP_Bypass )
   END_RUNG wire#w3
   RUNG wire#w1
      I_Contact( "General_Blend".CIP_Bypass )
      wire#w4
      Contact( "CIP_to_Mix".CIP_Supply_On."Buffer Cluster 2"."T-68.00_CIP_Supply_ON" )
      wire#w5
      Coil( "BFT-68"."CIP Supply ON" )
   END_RUNG
   RUNG wire#w4
      Contact( "CIP_to_Mix".CIP_Supply_On."Buffer Cluster 2"."T67&T68_CIP_LineToPasteur_Supply_ON" )
   END_RUNG wire#w5
   RUNG wire#w1
      Contact( "General_Blend".CIP_Bypass )
   END_RUNG wire#w5
   RUNG wire#w1
      I_Contact( "General_Blend".CIP_Bypass )
      wire#w6
      Contact( "CIP_to_Mix".CIP_Complete."Buffer Cluster 2"."T-68.00_CIP_Complete" )
      wire#w7
      Coil( "BFT-68"."CIP Complete" )
   END_RUNG
   RUNG wire#w6
      Contact( "CIP_to_Mix".CIP_Complete."Buffer Cluster 2"."T67&T68_CIP_LineToPasteur_Complete" )
   END_RUNG wire#w7
   // the same network as SCL:
   "BFT-68"."CIP Req OK" := "AlwaysTRUE" AND ((NOT "General_Blend".CIP_Bypass AND ("CIP_to_Mix".CIP_RequestOK."Buffer Cluster 2"."T-68.00_CIP_RequestOK" OR "CIP_to_Mix".CIP_RequestOK."Buffer Cluster 2"."T67&T68_CIP_LineToPasteur_RequestOK")) OR "General_Blend".CIP_Bypass);
   "BFT-68"."CIP Supply ON" := "AlwaysTRUE" AND ((NOT "General_Blend".CIP_Bypass AND ("CIP_to_Mix".CIP_Supply_On."Buffer Cluster 2"."T-68.00_CIP_Supply_ON" OR "CIP_to_Mix".CIP_Supply_On."Buffer Cluster 2"."T67&T68_CIP_LineToPasteur_Supply_ON")) OR "General_Blend".CIP_Bypass);
   "BFT-68"."CIP Complete" := "AlwaysTRUE" AND NOT "General_Blend".CIP_Bypass AND ("CIP_to_Mix".CIP_Complete."Buffer Cluster 2"."T-68.00_CIP_Complete" OR "CIP_to_Mix".CIP_Complete."Buffer Cluster 2"."T67&T68_CIP_LineToPasteur_Complete");
END_REGION

REGION Network 32: CIP Enable and CIP Line Open for Blending Cluster Line 1 Line 3
   RUNG wire#powerrail
      Contact( "AlwaysTRUE" )
      wire#w1
      I_Contact( "BFT-61".state.Inloading )
      Contact( "General_Blend".Blend_Cluster1.CIP_Line3."CIP Request" )
      Coil( "General Buffer"."CIP Enable".Cluster1_Line3 )
   END_RUNG
   RUNG wire#w1
      Contact( "General Buffer"."CIP Enable".Cluster1_Line3 )
      Contact( "IO_Valve_Buffer_DB"."AV-62.06".FB_OPEN )
      Coil( "General Buffer"."CIP Line Open".Cluster1_Line3 )
   END_RUNG
   // the same network as SCL:
   "General Buffer"."CIP Enable".Cluster1_Line3 := "AlwaysTRUE" AND NOT "BFT-61".state.Inloading AND "General_Blend".Blend_Cluster1.CIP_Line3."CIP Request";
   "General Buffer"."CIP Line Open".Cluster1_Line3 := "AlwaysTRUE" AND "General Buffer"."CIP Enable".Cluster1_Line3 AND "IO_Valve_Buffer_DB"."AV-62.06".FB_OPEN;
END_REGION

REGION Network 33: CIP Enable and CIP Line Open for Blending Cluster Line 2 Line 1
   RUNG wire#powerrail
      Contact( "AlwaysTRUE" )
      wire#w1
      I_Contact( "BFT-64".state.Inloading )
      Contact( "General_Blend".Blend_Cluster2.CIP_Line1."CIP Request" )
      Coil( "General Buffer"."CIP Enable".Cluster2_Line1 )
   END_RUNG
   RUNG wire#w1
      Contact( "General Buffer"."CIP Enable".Cluster2_Line1 )
      Contact( "IO_Valve_Buffer_DB"."AV-64.06".FB_OPEN )
      Coil( "General Buffer"."CIP Line Open".Cluster2_Line1 )
   END_RUNG
   // the same network as SCL:
   "General Buffer"."CIP Enable".Cluster2_Line1 := "AlwaysTRUE" AND NOT "BFT-64".state.Inloading AND "General_Blend".Blend_Cluster2.CIP_Line1."CIP Request";
   "General Buffer"."CIP Line Open".Cluster2_Line1 := "AlwaysTRUE" AND "General Buffer"."CIP Enable".Cluster2_Line1 AND "IO_Valve_Buffer_DB"."AV-64.06".FB_OPEN;
END_REGION

REGION Network 34: CIP Enable and CIP Line Open for Blending Cluster Line 2 Line 2
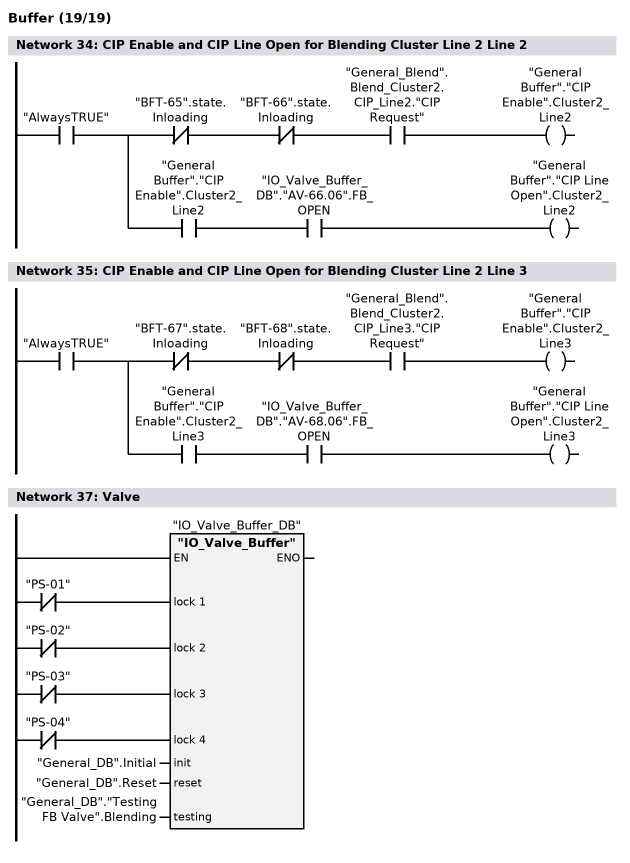
   RUNG wire#powerrail
      Contact( "AlwaysTRUE" )
      wire#w1
      I_Contact( "BFT-65".state.Inloading )
      I_Contact( "BFT-66".state.Inloading )
      Contact( "General_Blend".Blend_Cluster2.CIP_Line2."CIP Request" )
      Coil( "General Buffer"."CIP Enable".Cluster2_Line2 )
   END_RUNG
   RUNG wire#w1
      Contact( "General Buffer"."CIP Enable".Cluster2_Line2 )
      Contact( "IO_Valve_Buffer_DB"."AV-66.06".FB_OPEN )
      Coil( "General Buffer"."CIP Line Open".Cluster2_Line2 )
   END_RUNG
   // the same network as SCL:
   "General Buffer"."CIP Enable".Cluster2_Line2 := "AlwaysTRUE" AND NOT "BFT-65".state.Inloading AND NOT "BFT-66".state.Inloading AND "General_Blend".Blend_Cluster2.CIP_Line2."CIP Request";
   "General Buffer"."CIP Line Open".Cluster2_Line2 := "AlwaysTRUE" AND "General Buffer"."CIP Enable".Cluster2_Line2 AND "IO_Valve_Buffer_DB"."AV-66.06".FB_OPEN;
END_REGION

REGION Network 35: CIP Enable and CIP Line Open for Blending Cluster Line 2 Line 3
   RUNG wire#powerrail
      Contact( "AlwaysTRUE" )
      wire#w1
      I_Contact( "BFT-67".state.Inloading )
      I_Contact( "BFT-68".state.Inloading )
      Contact( "General_Blend".Blend_Cluster2.CIP_Line3."CIP Request" )
      Coil( "General Buffer"."CIP Enable".Cluster2_Line3 )
   END_RUNG
   RUNG wire#w1
      Contact( "General Buffer"."CIP Enable".Cluster2_Line3 )
      Contact( "IO_Valve_Buffer_DB"."AV-68.06".FB_OPEN )
      Coil( "General Buffer"."CIP Line Open".Cluster2_Line3 )
   END_RUNG
   // the same network as SCL:
   "General Buffer"."CIP Enable".Cluster2_Line3 := "AlwaysTRUE" AND NOT "BFT-67".state.Inloading AND NOT "BFT-68".state.Inloading AND "General_Blend".Blend_Cluster2.CIP_Line3."CIP Request";
   "General Buffer"."CIP Line Open".Cluster2_Line3 := "AlwaysTRUE" AND "General Buffer"."CIP Enable".Cluster2_Line3 AND "IO_Valve_Buffer_DB"."AV-68.06".FB_OPEN;
END_REGION

REGION Network 37: Valve
   RUNG wire#powerrail
      "IO_Valve_Buffer_DB"("lock 1" := wire#w1, "lock 2" := wire#w2, "lock 3" := wire#w3, "lock 4" := wire#w4, init := "General_DB".Initial, reset := "General_DB".Reset, testing := "General_DB"."Testing FB Valve".Blending)
   END_RUNG
   RUNG wire#powerrail
      I_Contact( "PS-01" )
   END_RUNG wire#w1
   RUNG wire#powerrail
      I_Contact( "PS-02" )
   END_RUNG wire#w2
   RUNG wire#powerrail
      I_Contact( "PS-03" )
   END_RUNG wire#w3
   RUNG wire#powerrail
      I_Contact( "PS-04" )
   END_RUNG wire#w4
   // the same network as SCL:
   "IO_Valve_Buffer_DB"("lock 1" := NOT "PS-01",   // "IO_Valve_Buffer"
                        "lock 2" := NOT "PS-02",
                        "lock 3" := NOT "PS-03",
                        "lock 4" := NOT "PS-04",
                        init := "General_DB".Initial,
                        reset := "General_DB".Reset,
                        testing := "General_DB"."Testing FB Valve".Blending);
END_REGION
END_FUNCTION

FUNCTION_BLOCK "Buffer_Tank"   // FB110, LAD
{ S7_Optimized_Access := 'TRUE' }
VERSION : 0.1
// stored: AutoNumber false, IsIECCheckEnabled false, IsRetainMemResEnabled false, MemoryReserve 100, SetENOAutomatically false, UDAEnableTagReadback false
   VAR_INPUT
      IN_LT01 : Real;
      "Tank w Circulation" : Bool;
      AlarmProd_pasteur : Bool;
      HighLevel_pasteur : Bool;
      IN_FBAV_Inload : Bool;
      IN_FBAV_CIP_Tank : Bool;
      IN_FBAV_CIP_Line : Bool;
      IN_FBAV_Outlet : Bool;
      IN_FBAV_Transfer : Bool;
      IN_FBP_Transfer : Bool;
      IN_FBXA : Bool;
      IN_FBP_Circulation : Bool;
      IN_Product_Ready : Bool;
      IN_Product_TransferOnProg : Bool;
      "Inload Busy" : Bool;
      "CIP Pulse" : Bool;
      "CIP Req OK" : Bool;
      "CIP Supply ON" : Bool;
      "CIP In Progress" : Bool;
      "CIP Complete" : Bool;
      "CIP Busy" : Bool;
   END_VAR
   VAR_OUTPUT
      Out_AV_Inload : Bool;
      Out_AV_Drain_In : Bool;
      Out_AV_CIP_Tank : Bool;
      Out_AV_CIP_Line : Bool;
      Out_AV_Outlet : Bool;
      Out_AV_Transfer : Bool;
      Out_P_Transfer : Bool;
      Out_P_Transfer_SP : Real;
      Out_XA : Bool;
      Out_XA_SP : Real;
      Out_P_Circulation : Bool;
      Out_Prod_Req : Bool;
      Out_Prod_LineOpen : Bool;
      Out_CIP_Tank_Req : Bool;
      Out_CIP_Line_Req : Bool;
      Out_CIP_Tank_LineOpen : Bool;
      Out_CIP_Line_LineOpen : Bool;
   END_VAR
   VAR
      cmd : Struct
         Inload : Bool;
         Drain_In : Bool;
         Ready_for_Transfer : Bool;
         CIP_Tank : Bool;
         CIP_Line : Bool;
         Agitator_Mode : Bool;
         Agitator_Man_OnOff : Bool;
         Agitator_SpeedMode : Bool;
         Circulation : Bool;
      END_STRUCT;
   END_VAR
   VAR RETAIN
      param : Struct
         L_Lo_Lim : Real;
         L_Hi_Lim : Real := 100.0;
         L_Hys : Real := 2.0;
         "Circulation Level" : Real := 20.0;
         SP_Level_HL : Real := 100.0;
         SP_Level_ML : Real := 80.0;
         SP_Level_LL : Real := 10.0;
         DrainIn : DInt := 10;
         SP_Pump_Transfer : Real := 80.0;
         SP_Pump_CIP : Real := 80.0;
         SP_Agitator : Real := 50.0;
         SP_Level_Agi_ON1 : Real := 20.0;
         SP_Level_Agi_OFF1 : Real := 49.0;
         SP_Level_Agi_ON2 : Real := 50.0;
         SP_Level_Agi_OFF2 : Real := 64.0;
         SP_Level_Agi_ON3 : Real := 65.0;
         "CIP Ret On" : Real := 5.0;
         "CIP Ret Off" : Real;
      END_STRUCT;
   END_VAR
   VAR
      state : Struct
         "Tank LL" : Bool;
         "Tank ML" : Bool;
         "Tank HL" : Bool;
         "Tank CIP En" : Bool;
         "Tank CIP" : Bool;
         "Line CIP En" : Bool;
         "Line CIP" : Bool;
         "Ready for Transfer En" : Bool;
         "Ready for Transfer" : Bool;
         Inloading : Bool;
         "Inload En" : Bool;
         L_Agi_ON1 : Bool;
         L_Agi_ON2 : Bool;
         L_Agi_ON3 : Bool;
         Tank_Circulation : Bool;
         "Circulation Enable" : Bool;
         Circulation : Bool;
         "Transfer on Prog" : Bool;
         "CIP Return On" : Bool;
         "CIP Req" : Bool;
      END_STRUCT;
      alwaysOn : Bool;
      L_Hys_Abs : Real;
      Hys_Level_LL : Real;
      Hys_Level_ML : Real;
      Hys_Level_HL : Real;
      Hys_Level_Circ : Real;
   END_VAR
   VAR DB_SPECIFIC
      r : Struct
         PosE1 : Bool;
         PosE2 : Bool;
         PosE3 : Bool;
         PosE4 : Bool;
         PosE5 : Bool;
         PosE6 : Bool;
         PosE7 : Bool;
         PosE8 : Bool;
         PosE9 : Bool;
         PosE10 : Bool;
         PosE11 : Bool;
         PosE12 : Bool;
         PosE13 : Bool;
         PosE14 : Bool;
         PosE15 : Bool;
         PosE16 : Bool;
         PosE17 : Bool;
         PosE18 : Bool;
         PosE19 : Bool;
         PosE20 : Bool;
         PosE21 : Bool;
         PosE22 : Bool;
         PosE23 : Bool;
         PosE24 : Bool;
         PosE25 : Bool;
         PosE26 : Bool;
         PosE27 : Bool;
         PosE28 : Bool;
         PosE29 : Bool;
         PosE30 : Bool;
         PosE31 : Bool;
         PosE32 : Bool;
      END_STRUCT;
      Actuator : Struct
         AV_Inload : Bool;
         AV_Drain_In : Bool;
         AV_Outlet : Bool;
         AV_Transfer : Bool;
         AV_CIP_Tank : Bool;
         AV_CIP_Line : Bool;
         P_Transfer : Bool;
         P_CIP : Bool;
         Agitator_level : Bool;
      END_STRUCT;
   END_VAR
   VAR
      DrainIn_OnTime : TON_TIME;
      DrainIn_OffTime : TOF_TIME;
      InloadAV_OffTime : TOF_TIME;
      DrainIn_MS : DInt;
      L_AgiTim : TON_TIME;
   END_VAR
   VAR_TEMP   // added for the SCL form of the ladder/FBD networks
      _w1 : Bool;
      _w2 : Bool;
      _w3 : Bool;
   END_VAR
BEGIN

REGION Network 1: always On
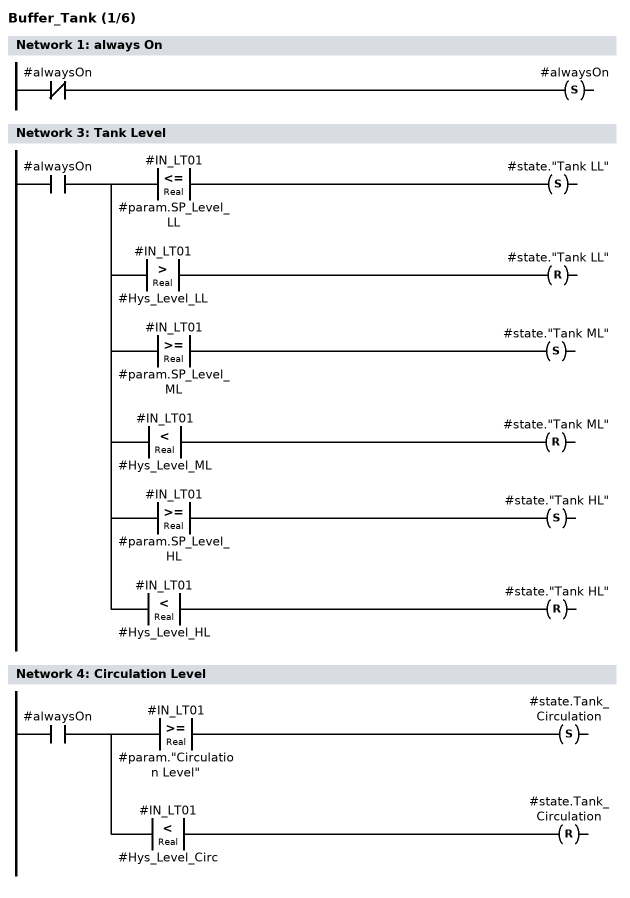
   RUNG wire#powerrail
      I_Contact( #alwaysOn )
      S_Coil( #alwaysOn )
   END_RUNG
   // the same network as SCL:
   IF NOT #alwaysOn THEN #alwaysOn := TRUE; END_IF;
END_REGION

NETWORK
TITLE = Hys Calculation
//Level Hys Absolute
      L     #param.L_Hi_Lim;
      L     #param.L_Lo_Lim;
      -R;
      L     100.0;
      /R;
      L     #param.L_Hys;
      *R;
      T     #L_Hys_Abs;
//Tank High Level
      L     #param.SP_Level_HL;
      L     #L_Hys_Abs;
      -R;
      T     #Hys_Level_HL;
//Tank Mid Level
      L     #param.SP_Level_ML;
      L     #L_Hys_Abs;
      -R;
      T     #Hys_Level_ML;
//Tank Low Level
      L     #param.SP_Level_LL;
      L     #L_Hys_Abs;
      +R;
      T     #Hys_Level_LL;
//Level Circulation
      L     #param."Circulation Level";
      L     #L_Hys_Abs;
      -R;
      T     #Hys_Level_Circ;



REGION Network 3: Tank Level
   RUNG wire#powerrail
      Contact( #alwaysOn )
      wire#w1
      { S7_Templates := "SrcType := Real" } LE_Contact(in1 := #IN_LT01, in2 := #param.SP_Level_LL)
      S_Coil( #state."Tank LL" )
   END_RUNG
   RUNG wire#w1
      { S7_Templates := "SrcType := Real" } GT_Contact(in1 := #IN_LT01, in2 := #Hys_Level_LL)
      R_Coil( #state."Tank LL" )
   END_RUNG
   RUNG wire#w1
      { S7_Templates := "SrcType := Real" } GE_Contact(in1 := #IN_LT01, in2 := #param.SP_Level_ML)
      S_Coil( #state."Tank ML" )
   END_RUNG
   RUNG wire#w1
      { S7_Templates := "SrcType := Real" } LT_Contact(in1 := #IN_LT01, in2 := #Hys_Level_ML)
      R_Coil( #state."Tank ML" )
   END_RUNG
   RUNG wire#w1
      { S7_Templates := "SrcType := Real" } GE_Contact(in1 := #IN_LT01, in2 := #param.SP_Level_HL)
      S_Coil( #state."Tank HL" )
   END_RUNG
   RUNG wire#w1
      { S7_Templates := "SrcType := Real" } LT_Contact(in1 := #IN_LT01, in2 := #Hys_Level_HL)
      R_Coil( #state."Tank HL" )
   END_RUNG
   // the same network as SCL:
   IF #alwaysOn AND (#IN_LT01 <= #param.SP_Level_LL) THEN #state."Tank LL" := TRUE; END_IF;
   IF #alwaysOn AND (#IN_LT01 > #Hys_Level_LL) THEN #state."Tank LL" := FALSE; END_IF;
   IF #alwaysOn AND (#IN_LT01 >= #param.SP_Level_ML) THEN #state."Tank ML" := TRUE; END_IF;
   IF #alwaysOn AND (#IN_LT01 < #Hys_Level_ML) THEN #state."Tank ML" := FALSE; END_IF;
   IF #alwaysOn AND (#IN_LT01 >= #param.SP_Level_HL) THEN #state."Tank HL" := TRUE; END_IF;
   IF #alwaysOn AND (#IN_LT01 < #Hys_Level_HL) THEN #state."Tank HL" := FALSE; END_IF;
END_REGION

REGION Network 4: Circulation Level
   RUNG wire#powerrail
      Contact( #alwaysOn )
      wire#w1
      { S7_Templates := "SrcType := Real" } GE_Contact(in1 := #IN_LT01, in2 := #param."Circulation Level")
      S_Coil( #state.Tank_Circulation )
   END_RUNG
   RUNG wire#w1
      { S7_Templates := "SrcType := Real" } LT_Contact(in1 := #IN_LT01, in2 := #Hys_Level_Circ)
      R_Coil( #state.Tank_Circulation )
   END_RUNG
   // the same network as SCL:
   IF #alwaysOn AND (#IN_LT01 >= #param."Circulation Level") THEN #state.Tank_Circulation := TRUE; END_IF;
   IF #alwaysOn AND (#IN_LT01 < #Hys_Level_Circ) THEN #state.Tank_Circulation := FALSE; END_IF;
END_REGION

REGION Network 5: Agitator Level ON-OFF
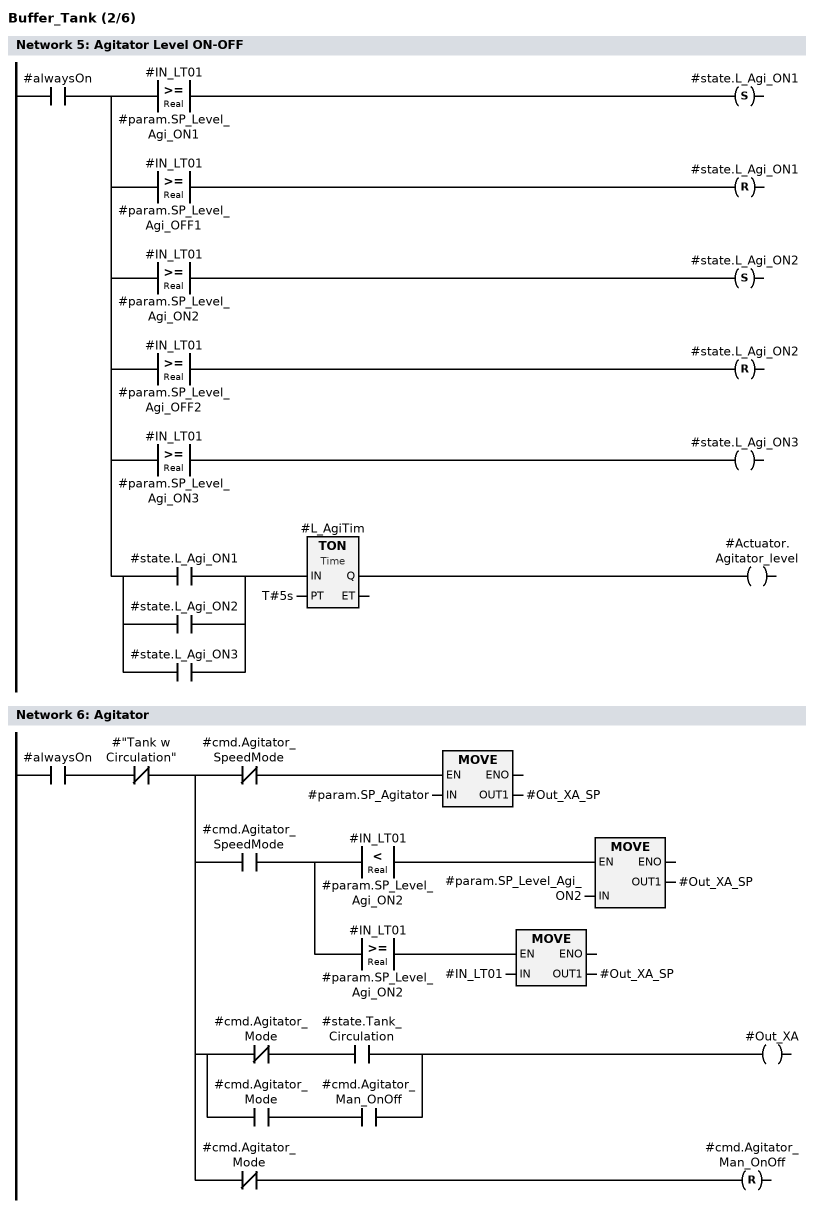
   RUNG wire#powerrail
      Contact( #alwaysOn )
      wire#w1
      { S7_Templates := "SrcType := Real" } GE_Contact(in1 := #IN_LT01, in2 := #param.SP_Level_Agi_ON1)
      S_Coil( #state.L_Agi_ON1 )
   END_RUNG
   RUNG wire#w1
      { S7_Templates := "SrcType := Real" } GE_Contact(in1 := #IN_LT01, in2 := #param.SP_Level_Agi_OFF1)
      R_Coil( #state.L_Agi_ON1 )
   END_RUNG
   RUNG wire#w1
      { S7_Templates := "SrcType := Real" } GE_Contact(in1 := #IN_LT01, in2 := #param.SP_Level_Agi_ON2)
      S_Coil( #state.L_Agi_ON2 )
   END_RUNG
   RUNG wire#w1
      { S7_Templates := "SrcType := Real" } GE_Contact(in1 := #IN_LT01, in2 := #param.SP_Level_Agi_OFF2)
      R_Coil( #state.L_Agi_ON2 )
   END_RUNG
   RUNG wire#w1
      { S7_Templates := "SrcType := Real" } GE_Contact(in1 := #IN_LT01, in2 := #param.SP_Level_Agi_ON3)
      Coil( #state.L_Agi_ON3 )
   END_RUNG
   RUNG wire#w1
      Contact( #state.L_Agi_ON1 )
      wire#w2
      { S7_Templates := "time_type := Time" } #L_AgiTim.TON(pt := T#5s, et =>)
      Coil( #Actuator.Agitator_level )
   END_RUNG
   RUNG wire#w1
      Contact( #state.L_Agi_ON2 )
   END_RUNG wire#w2
   RUNG wire#w1
      Contact( #state.L_Agi_ON3 )
   END_RUNG wire#w2
   // the same network as SCL:
   IF #alwaysOn AND (#IN_LT01 >= #param.SP_Level_Agi_ON1) THEN #state.L_Agi_ON1 := TRUE; END_IF;
   IF #alwaysOn AND (#IN_LT01 >= #param.SP_Level_Agi_OFF1) THEN #state.L_Agi_ON1 := FALSE; END_IF;
   IF #alwaysOn AND (#IN_LT01 >= #param.SP_Level_Agi_ON2) THEN #state.L_Agi_ON2 := TRUE; END_IF;
   IF #alwaysOn AND (#IN_LT01 >= #param.SP_Level_Agi_OFF2) THEN #state.L_Agi_ON2 := FALSE; END_IF;
   #state.L_Agi_ON3 := #alwaysOn AND (#IN_LT01 >= #param.SP_Level_Agi_ON3);
   #L_AgiTim(IN := #alwaysOn AND (#state.L_Agi_ON1 OR #state.L_Agi_ON2 OR #state.L_Agi_ON3), PT := T#5s);   // TON
   #Actuator.Agitator_level := #L_AgiTim.Q;
END_REGION

REGION Network 6: Agitator
   RUNG wire#powerrail
      Contact( #alwaysOn )
      I_Contact( #"Tank w Circulation" )
      wire#w1
      I_Contact( #cmd.Agitator_SpeedMode )
      Move(in := #param.SP_Agitator, out1 => #Out_XA_SP)
   END_RUNG
   RUNG wire#w1
      Contact( #cmd.Agitator_SpeedMode )
      wire#w2
      { S7_Templates := "SrcType := Real" } LT_Contact(in1 := #IN_LT01, in2 := #param.SP_Level_Agi_ON2)
      Move(in := #param.SP_Level_Agi_ON2, out1 => #Out_XA_SP)
   END_RUNG
   RUNG wire#w2
      { S7_Templates := "SrcType := Real" } GE_Contact(in1 := #IN_LT01, in2 := #param.SP_Level_Agi_ON2)
      Move(in := #IN_LT01, out1 => #Out_XA_SP)
   END_RUNG
   RUNG wire#w1
      I_Contact( #cmd.Agitator_Mode )
      Contact( #state.Tank_Circulation )
      wire#w3
      Coil( #Out_XA )
   END_RUNG
   RUNG wire#w1
      Contact( #cmd.Agitator_Mode )
      Contact( #cmd.Agitator_Man_OnOff )
   END_RUNG wire#w3
   RUNG wire#w1
      I_Contact( #cmd.Agitator_Mode )
      R_Coil( #cmd.Agitator_Man_OnOff )
   END_RUNG
   // the same network as SCL:
   #_w1 := #alwaysOn AND NOT #"Tank w Circulation";
   IF #_w1 AND NOT #cmd.Agitator_SpeedMode THEN #Out_XA_SP := #param.SP_Agitator; END_IF;
   #_w2 := #_w1 AND #cmd.Agitator_SpeedMode;
   IF #_w2 AND (#IN_LT01 < #param.SP_Level_Agi_ON2) THEN #Out_XA_SP := #param.SP_Level_Agi_ON2; END_IF;
   IF #_w2 AND (#IN_LT01 >= #param.SP_Level_Agi_ON2) THEN #Out_XA_SP := #IN_LT01; END_IF;
   #Out_XA := #_w1 AND ((NOT #cmd.Agitator_Mode AND #state.Tank_Circulation) OR (#cmd.Agitator_Mode AND #cmd.Agitator_Man_OnOff));
   IF #_w1 AND NOT #cmd.Agitator_Mode THEN #cmd.Agitator_Man_OnOff := FALSE; END_IF;
END_REGION

REGION Network 7: Circulation
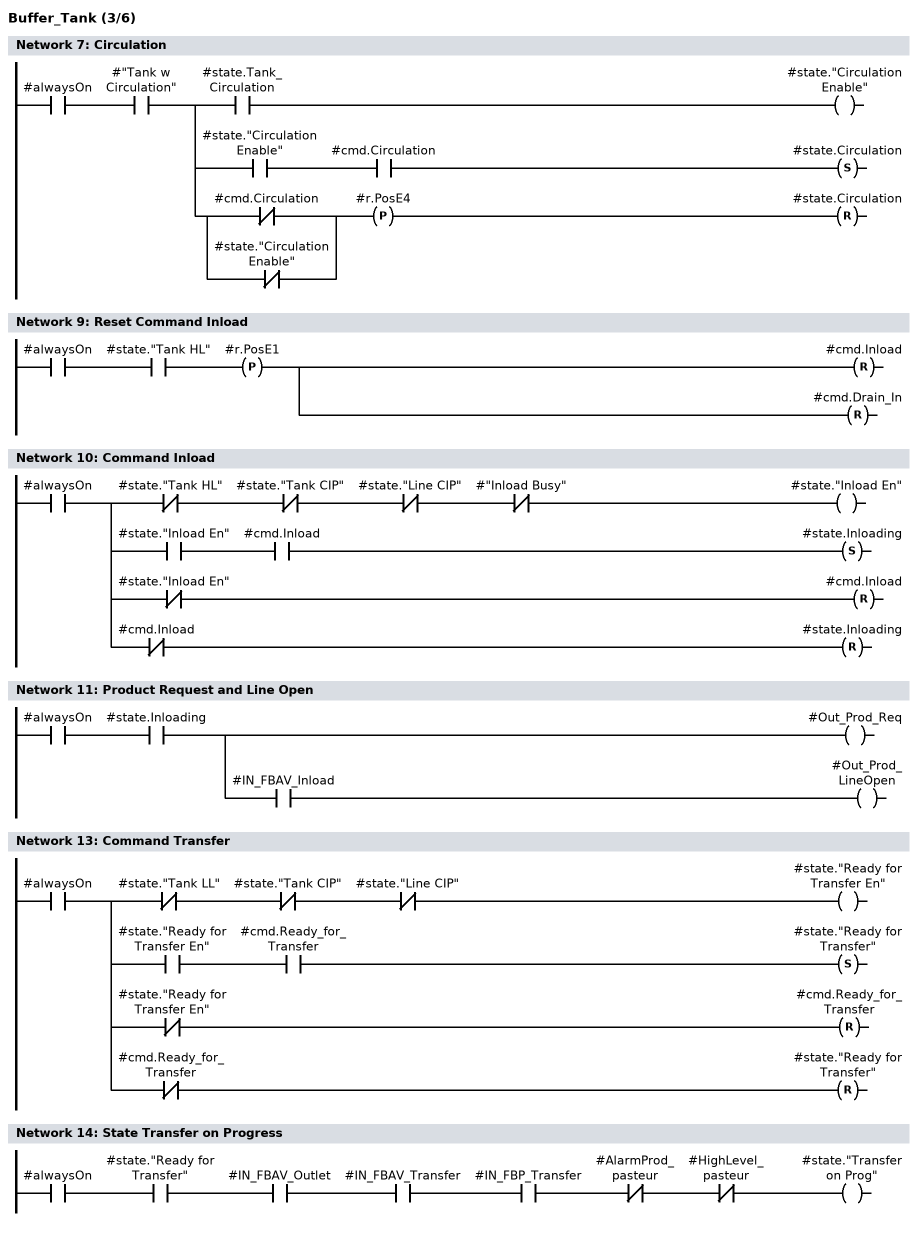
   RUNG wire#powerrail
      Contact( #alwaysOn )
      Contact( #"Tank w Circulation" )
      wire#w1
      Contact( #state.Tank_Circulation )
      Coil( #state."Circulation Enable" )
   END_RUNG
   RUNG wire#w1
      Contact( #state."Circulation Enable" )
      Contact( #cmd.Circulation )
      S_Coil( #state.Circulation )
   END_RUNG
   RUNG wire#w1
      I_Contact( #cmd.Circulation )
      wire#w2
      P_Trig( #r.PosE4 )
      R_Coil( #state.Circulation )
   END_RUNG
   RUNG wire#w1
      I_Contact( #state."Circulation Enable" )
   END_RUNG wire#w2
   // the same network as SCL:
   #_w1 := #alwaysOn AND #"Tank w Circulation";
   #state."Circulation Enable" := #_w1 AND #state.Tank_Circulation;
   IF #_w1 AND #state."Circulation Enable" AND #cmd.Circulation THEN #state.Circulation := TRUE; END_IF;
   #_w2 := #_w1 AND (NOT #cmd.Circulation OR NOT #state."Circulation Enable");
   #_w3 := #_w2 AND NOT #r.PosE4;   // rising edge
   #r.PosE4 := #_w2;
   IF #_w3 THEN #state.Circulation := FALSE; END_IF;
END_REGION

REGION Network 9: Reset Command Inload
   RUNG wire#powerrail
      Contact( #alwaysOn )
      Contact( #state."Tank HL" )
      P_Trig( #r.PosE1 )
      wire#w1
      R_Coil( #cmd.Inload )
   END_RUNG
   RUNG wire#w1
      R_Coil( #cmd.Drain_In )
   END_RUNG
   // the same network as SCL:
   #_w1 := #alwaysOn AND #state."Tank HL";
   #_w2 := #_w1 AND NOT #r.PosE1;   // rising edge
   #r.PosE1 := #_w1;
   IF #_w2 THEN
       #cmd.Inload := FALSE;
       #cmd.Drain_In := FALSE;
   END_IF;
END_REGION

REGION Network 10: Command Inload
   RUNG wire#powerrail
      Contact( #alwaysOn )
      wire#w1
      I_Contact( #state."Tank HL" )
      I_Contact( #state."Tank CIP" )
      I_Contact( #state."Line CIP" )
      I_Contact( #"Inload Busy" )
      Coil( #state."Inload En" )
   END_RUNG
   RUNG wire#w1
      Contact( #state."Inload En" )
      Contact( #cmd.Inload )
      S_Coil( #state.Inloading )
   END_RUNG
   RUNG wire#w1
      I_Contact( #state."Inload En" )
      R_Coil( #cmd.Inload )
   END_RUNG
   RUNG wire#w1
      I_Contact( #cmd.Inload )
      R_Coil( #state.Inloading )
   END_RUNG
   // the same network as SCL:
   #state."Inload En" := #alwaysOn AND NOT #state."Tank HL" AND NOT #state."Tank CIP" AND NOT #state."Line CIP" AND NOT #"Inload Busy";
   IF #alwaysOn AND #state."Inload En" AND #cmd.Inload THEN #state.Inloading := TRUE; END_IF;
   IF #alwaysOn AND NOT #state."Inload En" THEN #cmd.Inload := FALSE; END_IF;
   IF #alwaysOn AND NOT #cmd.Inload THEN #state.Inloading := FALSE; END_IF;
END_REGION

REGION Network 11: Product Request and Line Open
   RUNG wire#powerrail
      Contact( #alwaysOn )
      Contact( #state.Inloading )
      wire#w1
      Coil( #Out_Prod_Req )
   END_RUNG
   RUNG wire#w1
      Contact( #IN_FBAV_Inload )
      Coil( #Out_Prod_LineOpen )
   END_RUNG
   // the same network as SCL:
   #Out_Prod_Req := #alwaysOn AND #state.Inloading;
   #Out_Prod_LineOpen := #Out_Prod_Req AND #IN_FBAV_Inload;
END_REGION

REGION Network 13: Command Transfer
   RUNG wire#powerrail
      Contact( #alwaysOn )
      wire#w1
      I_Contact( #state."Tank LL" )
      I_Contact( #state."Tank CIP" )
      I_Contact( #state."Line CIP" )
      Coil( #state."Ready for Transfer En" )
   END_RUNG
   RUNG wire#w1
      Contact( #state."Ready for Transfer En" )
      Contact( #cmd.Ready_for_Transfer )
      S_Coil( #state."Ready for Transfer" )
   END_RUNG
   RUNG wire#w1
      I_Contact( #state."Ready for Transfer En" )
      R_Coil( #cmd.Ready_for_Transfer )
   END_RUNG
   RUNG wire#w1
      I_Contact( #cmd.Ready_for_Transfer )
      R_Coil( #state."Ready for Transfer" )
   END_RUNG
   // the same network as SCL:
   #state."Ready for Transfer En" := #alwaysOn AND NOT #state."Tank LL" AND NOT #state."Tank CIP" AND NOT #state."Line CIP";
   IF #alwaysOn AND #state."Ready for Transfer En" AND #cmd.Ready_for_Transfer THEN
       #state."Ready for Transfer" := TRUE;
   END_IF;
   IF #alwaysOn AND NOT #state."Ready for Transfer En" THEN #cmd.Ready_for_Transfer := FALSE; END_IF;
   IF #alwaysOn AND NOT #cmd.Ready_for_Transfer THEN #state."Ready for Transfer" := FALSE; END_IF;
END_REGION

REGION Network 14: State Transfer on Progress
   RUNG wire#powerrail
      Contact( #alwaysOn )
      Contact( #state."Ready for Transfer" )
      Contact( #IN_FBAV_Outlet )
      Contact( #IN_FBAV_Transfer )
      Contact( #IN_FBP_Transfer )
      I_Contact( #AlarmProd_pasteur )
      I_Contact( #HighLevel_pasteur )
      Coil( #state."Transfer on Prog" )
   END_RUNG
   // the same network as SCL:
   #state."Transfer on Prog" := #alwaysOn AND #state."Ready for Transfer" AND #IN_FBAV_Outlet AND #IN_FBAV_Transfer AND #IN_FBP_Transfer AND NOT #AlarmProd_pasteur AND NOT #HighLevel_pasteur;
END_REGION

REGION Network 16: Command CIP
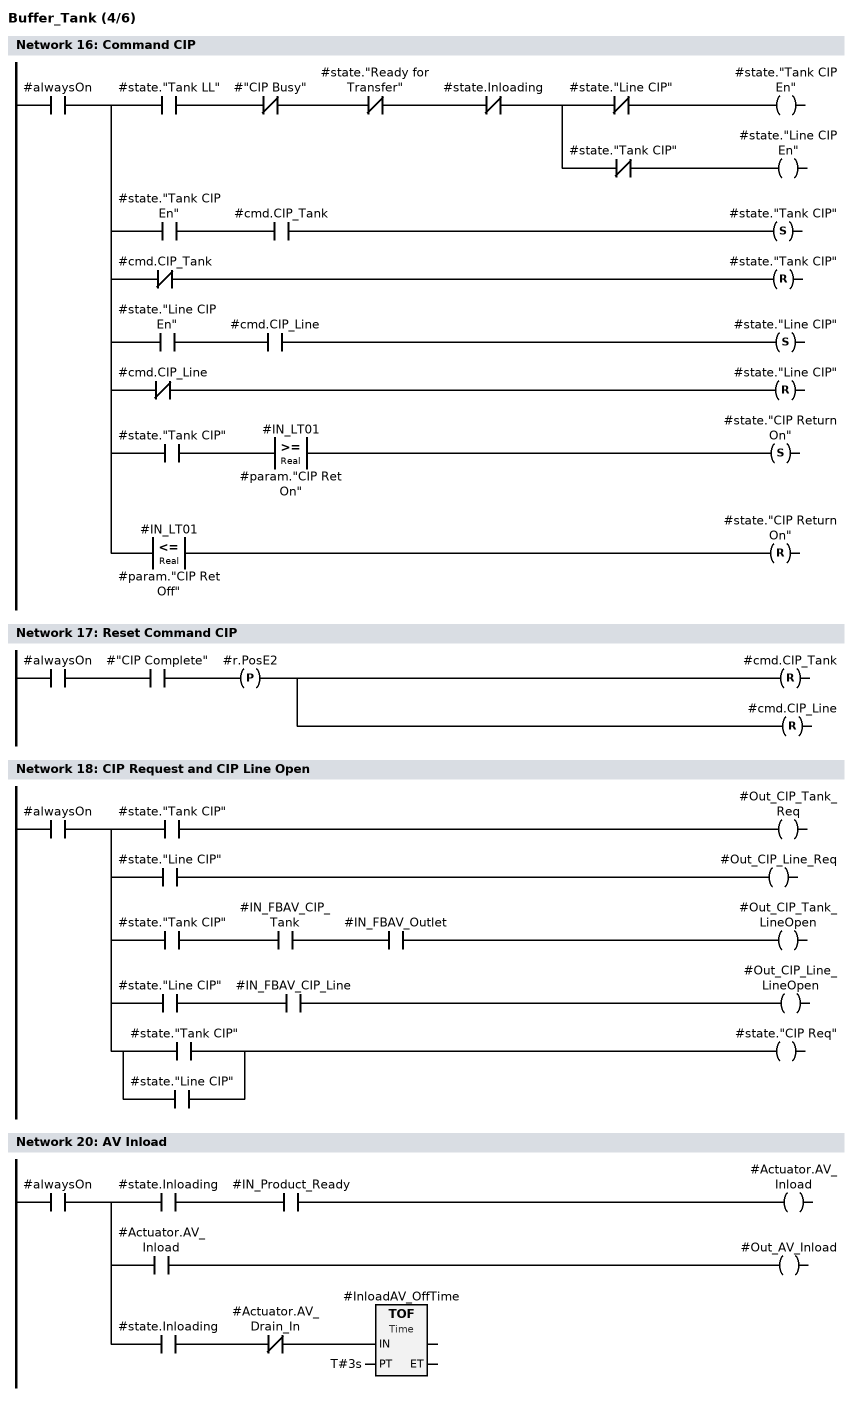
   RUNG wire#powerrail
      Contact( #alwaysOn )
      wire#w1
      Contact( #state."Tank LL" )
      I_Contact( #"CIP Busy" )
      I_Contact( #state."Ready for Transfer" )
      I_Contact( #state.Inloading )
      wire#w2
      I_Contact( #state."Line CIP" )
      Coil( #state."Tank CIP En" )
   END_RUNG
   RUNG wire#w2
      I_Contact( #state."Tank CIP" )
      Coil( #state."Line CIP En" )
   END_RUNG
   RUNG wire#w1
      Contact( #state."Tank CIP En" )
      Contact( #cmd.CIP_Tank )
      S_Coil( #state."Tank CIP" )
   END_RUNG
   RUNG wire#w1
      I_Contact( #cmd.CIP_Tank )
      R_Coil( #state."Tank CIP" )
   END_RUNG
   RUNG wire#w1
      Contact( #state."Line CIP En" )
      Contact( #cmd.CIP_Line )
      S_Coil( #state."Line CIP" )
   END_RUNG
   RUNG wire#w1
      I_Contact( #cmd.CIP_Line )
      R_Coil( #state."Line CIP" )
   END_RUNG
   RUNG wire#w1
      Contact( #state."Tank CIP" )
      { S7_Templates := "SrcType := Real" } GE_Contact(in1 := #IN_LT01, in2 := #param."CIP Ret On")
      S_Coil( #state."CIP Return On" )
   END_RUNG
   RUNG wire#w1
      { S7_Templates := "SrcType := Real" } LE_Contact(in1 := #IN_LT01, in2 := #param."CIP Ret Off")
      R_Coil( #state."CIP Return On" )
   END_RUNG
   // the same network as SCL:
   #_w1 := #alwaysOn AND #state."Tank LL" AND NOT #"CIP Busy" AND NOT #state."Ready for Transfer" AND NOT #state.Inloading;
   #state."Tank CIP En" := #_w1 AND NOT #state."Line CIP";
   #state."Line CIP En" := #_w1 AND NOT #state."Tank CIP";
   IF #alwaysOn AND #state."Tank CIP En" AND #cmd.CIP_Tank THEN #state."Tank CIP" := TRUE; END_IF;
   IF #alwaysOn AND NOT #cmd.CIP_Tank THEN #state."Tank CIP" := FALSE; END_IF;
   IF #alwaysOn AND #state."Line CIP En" AND #cmd.CIP_Line THEN #state."Line CIP" := TRUE; END_IF;
   IF #alwaysOn AND NOT #cmd.CIP_Line THEN #state."Line CIP" := FALSE; END_IF;
   IF #alwaysOn AND #state."Tank CIP" AND (#IN_LT01 >= #param."CIP Ret On") THEN
       #state."CIP Return On" := TRUE;
   END_IF;
   IF #alwaysOn AND (#IN_LT01 <= #param."CIP Ret Off") THEN #state."CIP Return On" := FALSE; END_IF;
END_REGION

REGION Network 17: Reset Command CIP
   RUNG wire#powerrail
      Contact( #alwaysOn )
      Contact( #"CIP Complete" )
      P_Trig( #r.PosE2 )
      wire#w1
      R_Coil( #cmd.CIP_Tank )
   END_RUNG
   RUNG wire#w1
      R_Coil( #cmd.CIP_Line )
   END_RUNG
   // the same network as SCL:
   #_w1 := #alwaysOn AND #"CIP Complete";
   #_w2 := #_w1 AND NOT #r.PosE2;   // rising edge
   #r.PosE2 := #_w1;
   IF #_w2 THEN
       #cmd.CIP_Tank := FALSE;
       #cmd.CIP_Line := FALSE;
   END_IF;
END_REGION

REGION Network 18: CIP Request and CIP Line Open
   RUNG wire#powerrail
      Contact( #alwaysOn )
      wire#w1
      Contact( #state."Tank CIP" )
      Coil( #Out_CIP_Tank_Req )
   END_RUNG
   RUNG wire#w1
      Contact( #state."Line CIP" )
      Coil( #Out_CIP_Line_Req )
   END_RUNG
   RUNG wire#w1
      Contact( #state."Tank CIP" )
      Contact( #IN_FBAV_CIP_Tank )
      Contact( #IN_FBAV_Outlet )
      Coil( #Out_CIP_Tank_LineOpen )
   END_RUNG
   RUNG wire#w1
      Contact( #state."Line CIP" )
      Contact( #IN_FBAV_CIP_Line )
      Coil( #Out_CIP_Line_LineOpen )
   END_RUNG
   RUNG wire#w1
      Contact( #state."Tank CIP" )
      wire#w2
      Coil( #state."CIP Req" )
   END_RUNG
   RUNG wire#w1
      Contact( #state."Line CIP" )
   END_RUNG wire#w2
   // the same network as SCL:
   #Out_CIP_Tank_Req := #alwaysOn AND #state."Tank CIP";
   #Out_CIP_Line_Req := #alwaysOn AND #state."Line CIP";
   #Out_CIP_Tank_LineOpen := #alwaysOn AND #state."Tank CIP" AND #IN_FBAV_CIP_Tank AND #IN_FBAV_Outlet;
   #Out_CIP_Line_LineOpen := #alwaysOn AND #state."Line CIP" AND #IN_FBAV_CIP_Line;
   #state."CIP Req" := #alwaysOn AND (#state."Tank CIP" OR #state."Line CIP");
END_REGION

REGION Network 20: AV Inload
   RUNG wire#powerrail
      Contact( #alwaysOn )
      wire#w1
      Contact( #state.Inloading )
      Contact( #IN_Product_Ready )
      Coil( #Actuator.AV_Inload )
   END_RUNG
   RUNG wire#w1
      Contact( #Actuator.AV_Inload )
      Coil( #Out_AV_Inload )
   END_RUNG
   RUNG wire#w1
      Contact( #state.Inloading )
      I_Contact( #Actuator.AV_Drain_In )
      { S7_Templates := "time_type := Time" } #InloadAV_OffTime.TOF(pt := T#3s, et =>)
   END_RUNG
   // the same network as SCL:
   #Actuator.AV_Inload := #alwaysOn AND #state.Inloading AND #IN_Product_Ready;
   #Out_AV_Inload := #alwaysOn AND #Actuator.AV_Inload;
   #InloadAV_OffTime(IN := #alwaysOn AND #state.Inloading AND NOT #Actuator.AV_Drain_In, PT := T#3s);   // TOF
END_REGION

REGION Network 21: AV Drain In
